REGION Network 10: Stack Door Common Monitoring#7
   RUNG wire#powerrail
      Contact( #TRUE )
      wire#w1
      Contact( "Safety.DataFromSafety".fDoorCoilStatus.anodeWasteDoorUnlock )
      wire#w2
      Coil( "Safetyinterface".StackDoor7.monitoring.DoorOpen )
   END_RUNG
   RUNG wire#w1
      I_Contact( "Safety.DataFromSafety".fDoorCoilStatus.anodeWasteDoorUnlock )
      Contact( "Safety.DataFromSafety".fDoorDrive.fDoor7.ackReq )
      I_Contact( "Global.Data".general.clock.cycle1000Msec )
      I_Contact( "Safety.DataFromSafety".fDoorSwitchStatus.anodeWasteDoorOpen )
   END_RUNG wire#w2
   RUNG wire#w1
      Contact( "Safety.DataFromSafety".fDoorCoilStatus.anodeWasteDoorUnlock )
      Coil( "Safetyinterface".StackDoor7.monitoring.DoorUnLock )
   END_RUNG
   RUNG wire#w1
      I_Contact( "Safety.DataFromSafety".fDoorCoilStatus.anodeWasteDoorUnlock )
      wire#w3
      I_Contact( "Safety.DataFromSafety".fDoorDrive.fDoor7.ackReq )
      wire#w4
      I_Contact( "Safety.DataFromSafety".fDoorSwitchStatus.anodeWasteDoorOpen )
      I_Contact( "Safetyinterface".StackDoor7.monitoring.DoorOpen )
      Coil( "Safetyinterface".StackDoor7.monitoring.DoorClose )
   END_RUNG
   RUNG wire#w3
      Contact( "Safety.DataFromSafety".fDoorDrive.fDoor7.ackReq )
      I_Contact( "Global.Data".general.clock.cycle1000Msec )
   END_RUNG wire#w4
   RUNG wire#w4
      Coil( "Safetyinterface".StackDoor7.monitoring.DoorLock )
   END_RUNG
   // the same network as SCL:
   "Safetyinterface".StackDoor7.monitoring.DoorOpen := #TRUE AND ("Safety.DataFromSafety".fDoorCoilStatus.anodeWasteDoorUnlock OR (NOT "Safety.DataFromSafety".fDoorCoilStatus.anodeWasteDoorUnlock AND "Safety.DataFromSafety".fDoorDrive.fDoor7.ackReq AND NOT "Global.Data".general.clock.cycle1000Msec AND NOT "Safety.DataFromSafety".fDoorSwitchStatus.anodeWasteDoorOpen));
   "Safetyinterface".StackDoor7.monitoring.DoorUnLock := #TRUE AND "Safety.DataFromSafety".fDoorCoilStatus.anodeWasteDoorUnlock;
   #_w1 := #TRUE AND NOT "Safety.DataFromSafety".fDoorCoilStatus.anodeWasteDoorUnlock AND (NOT "Safety.DataFromSafety".fDoorDrive.fDoor7.ackReq OR ("Safety.DataFromSafety".fDoorDrive.fDoor7.ackReq AND NOT "Global.Data".general.clock.cycle1000Msec));
   "Safetyinterface".StackDoor7.monitoring.DoorClose := #_w1 AND NOT "Safety.DataFromSafety".fDoorSwitchStatus.anodeWasteDoorOpen AND NOT "Safetyinterface".StackDoor7.monitoring.DoorOpen;
   "Safetyinterface".StackDoor7.monitoring.DoorLock := #_w1;
END_REGION

REGION Network 11: Stack Door Common Command#8
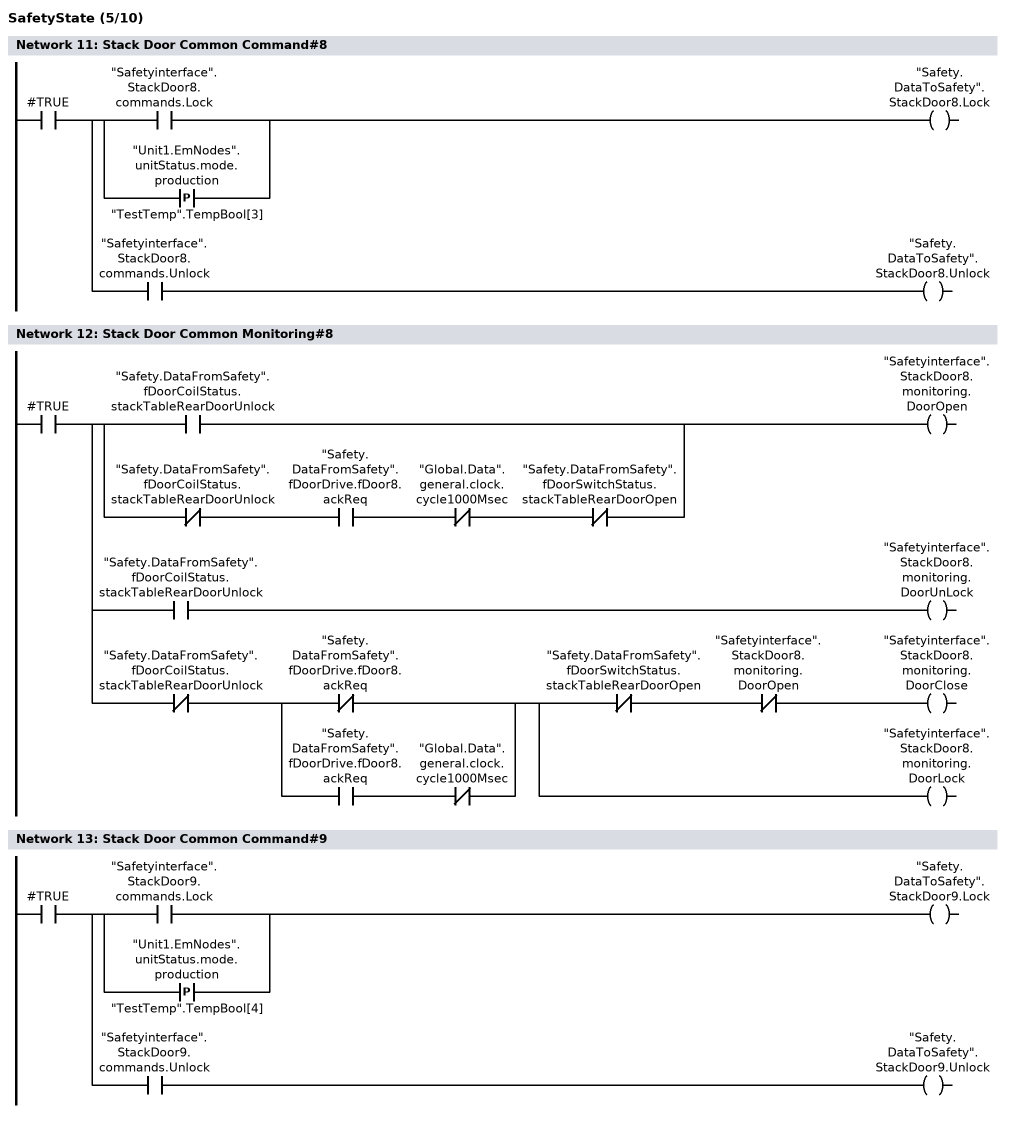
   RUNG wire#powerrail
      Contact( #TRUE )
      wire#w1
      Contact( "Safetyinterface".StackDoor8.commands.Lock )
      wire#w2
      Coil( "Safety.DataToSafety".StackDoor8.Lock )
   END_RUNG
   RUNG wire#w1
      P_Contact(operand := "Unit1.EmNodes".unitStatus.mode.production, bit := "TestTemp".TempBool[3])
   END_RUNG wire#w2
   RUNG wire#w1
      Contact( "Safetyinterface".StackDoor8.commands.Unlock )
      Coil( "Safety.DataToSafety".StackDoor8.Unlock )
   END_RUNG
   // the same network as SCL:
   #_w1 := #TRUE AND "Unit1.EmNodes".unitStatus.mode.production AND NOT "TestTemp".TempBool[3];   // rising edge of "Unit1.EmNodes".unitStatus.mode.production
   "TestTemp".TempBool[3] := "Unit1.EmNodes".unitStatus.mode.production;
   "Safety.DataToSafety".StackDoor8.Lock := (#TRUE AND "Safetyinterface".StackDoor8.commands.Lock) OR #_w1;
   "Safety.DataToSafety".StackDoor8.Unlock := #TRUE AND "Safetyinterface".StackDoor8.commands.Unlock;
END_REGION

REGION Network 12: Stack Door Common Monitoring#8
   RUNG wire#powerrail
      Contact( #TRUE )
      wire#w1
      Contact( "Safety.DataFromSafety".fDoorCoilStatus.stackTableRearDoorUnlock )
      wire#w2
      Coil( "Safetyinterface".StackDoor8.monitoring.DoorOpen )
   END_RUNG
   RUNG wire#w1
      I_Contact( "Safety.DataFromSafety".fDoorCoilStatus.stackTableRearDoorUnlock )
      Contact( "Safety.DataFromSafety".fDoorDrive.fDoor8.ackReq )
      I_Contact( "Global.Data".general.clock.cycle1000Msec )
      I_Contact( "Safety.DataFromSafety".fDoorSwitchStatus.stackTableRearDoorOpen )
   END_RUNG wire#w2
   RUNG wire#w1
      Contact( "Safety.DataFromSafety".fDoorCoilStatus.stackTableRearDoorUnlock )
      Coil( "Safetyinterface".StackDoor8.monitoring.DoorUnLock )
   END_RUNG
   RUNG wire#w1
      I_Contact( "Safety.DataFromSafety".fDoorCoilStatus.stackTableRearDoorUnlock )
      wire#w3
      I_Contact( "Safety.DataFromSafety".fDoorDrive.fDoor8.ackReq )
      wire#w4
      I_Contact( "Safety.DataFromSafety".fDoorSwitchStatus.stackTableRearDoorOpen )
      I_Contact( "Safetyinterface".StackDoor8.monitoring.DoorOpen )
      Coil( "Safetyinterface".StackDoor8.monitoring.DoorClose )
   END_RUNG
   RUNG wire#w3
      Contact( "Safety.DataFromSafety".fDoorDrive.fDoor8.ackReq )
      I_Contact( "Global.Data".general.clock.cycle1000Msec )
   END_RUNG wire#w4
   RUNG wire#w4
      Coil( "Safetyinterface".StackDoor8.monitoring.DoorLock )
   END_RUNG
   // the same network as SCL:
   "Safetyinterface".StackDoor8.monitoring.DoorOpen := #TRUE AND ("Safety.DataFromSafety".fDoorCoilStatus.stackTableRearDoorUnlock OR (NOT "Safety.DataFromSafety".fDoorCoilStatus.stackTableRearDoorUnlock AND "Safety.DataFromSafety".fDoorDrive.fDoor8.ackReq AND NOT "Global.Data".general.clock.cycle1000Msec AND NOT "Safety.DataFromSafety".fDoorSwitchStatus.stackTableRearDoorOpen));
   "Safetyinterface".StackDoor8.monitoring.DoorUnLock := #TRUE AND "Safety.DataFromSafety".fDoorCoilStatus.stackTableRearDoorUnlock;
   #_w1 := #TRUE AND NOT "Safety.DataFromSafety".fDoorCoilStatus.stackTableRearDoorUnlock AND (NOT "Safety.DataFromSafety".fDoorDrive.fDoor8.ackReq OR ("Safety.DataFromSafety".fDoorDrive.fDoor8.ackReq AND NOT "Global.Data".general.clock.cycle1000Msec));
   "Safetyinterface".StackDoor8.monitoring.DoorClose := #_w1 AND NOT "Safety.DataFromSafety".fDoorSwitchStatus.stackTableRearDoorOpen AND NOT "Safetyinterface".StackDoor8.monitoring.DoorOpen;
   "Safetyinterface".StackDoor8.monitoring.DoorLock := #_w1;
END_REGION

REGION Network 13: Stack Door Common Command#9
   RUNG wire#powerrail
      Contact( #TRUE )
      wire#w1
      Contact( "Safetyinterface".StackDoor9.commands.Lock )
      wire#w2
      Coil( "Safety.DataToSafety".StackDoor9.Lock )
   END_RUNG
   RUNG wire#w1
      P_Contact(operand := "Unit1.EmNodes".unitStatus.mode.production, bit := "TestTemp".TempBool[4])
   END_RUNG wire#w2
   RUNG wire#w1
      Contact( "Safetyinterface".StackDoor9.commands.Unlock )
      Coil( "Safety.DataToSafety".StackDoor9.Unlock )
   END_RUNG
   // the same network as SCL:
   #_w1 := #TRUE AND "Unit1.EmNodes".unitStatus.mode.production AND NOT "TestTemp".TempBool[4];   // rising edge of "Unit1.EmNodes".unitStatus.mode.production
   "TestTemp".TempBool[4] := "Unit1.EmNodes".unitStatus.mode.production;
   "Safety.DataToSafety".StackDoor9.Lock := (#TRUE AND "Safetyinterface".StackDoor9.commands.Lock) OR #_w1;
   "Safety.DataToSafety".StackDoor9.Unlock := #TRUE AND "Safetyinterface".StackDoor9.commands.Unlock;
END_REGION

REGION Network 14: Stack Door Common Monitoring#9
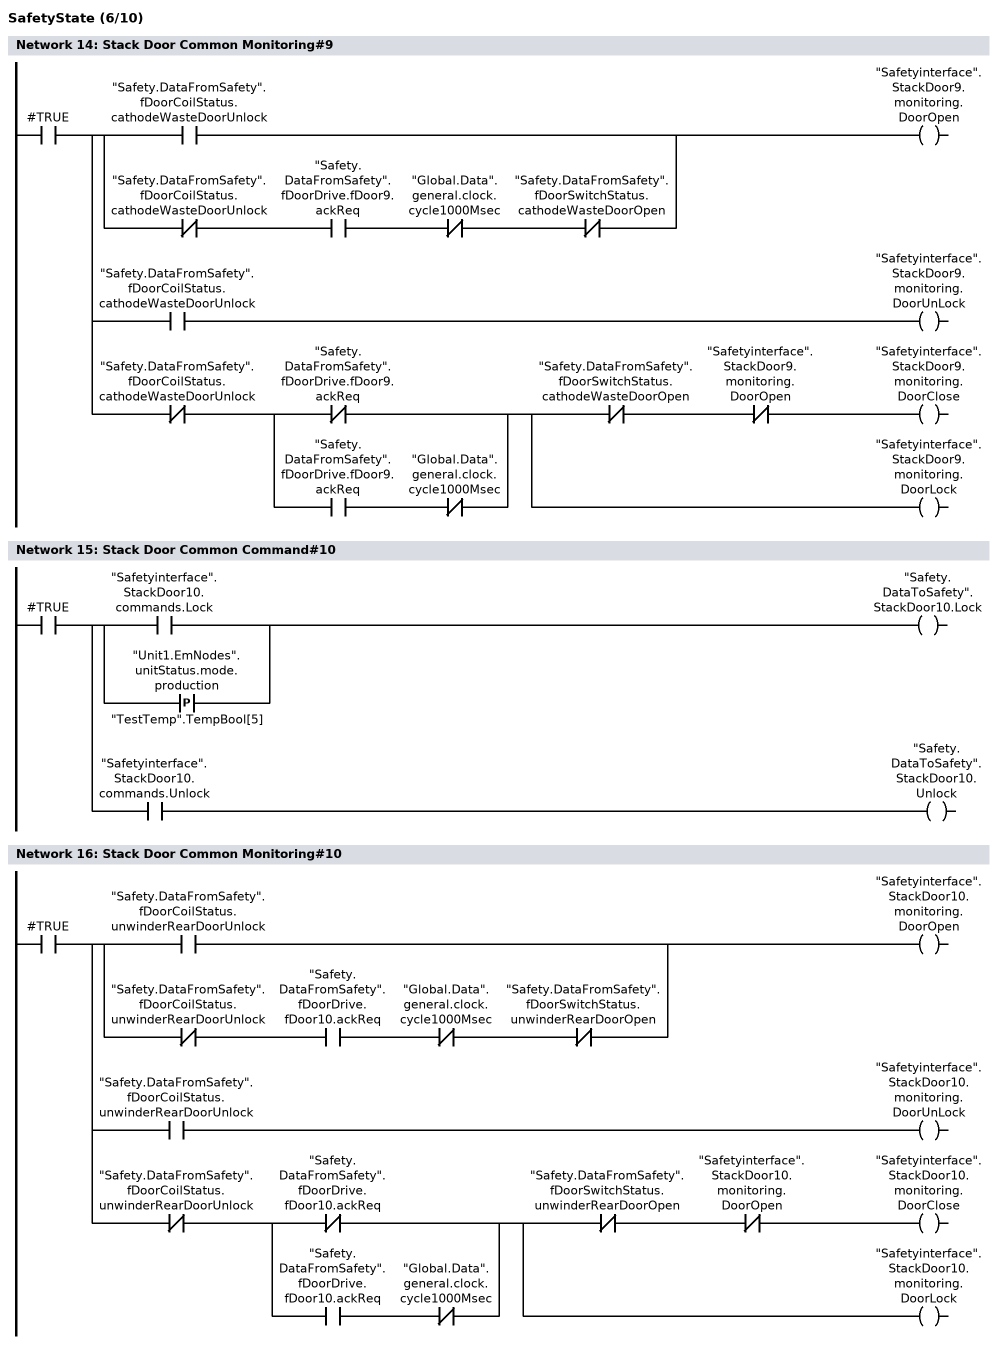
   RUNG wire#powerrail
      Contact( #TRUE )
      wire#w1
      Contact( "Safety.DataFromSafety".fDoorCoilStatus.cathodeWasteDoorUnlock )
      wire#w2
      Coil( "Safetyinterface".StackDoor9.monitoring.DoorOpen )
   END_RUNG
   RUNG wire#w1
      I_Contact( "Safety.DataFromSafety".fDoorCoilStatus.cathodeWasteDoorUnlock )
      Contact( "Safety.DataFromSafety".fDoorDrive.fDoor9.ackReq )
      I_Contact( "Global.Data".general.clock.cycle1000Msec )
      I_Contact( "Safety.DataFromSafety".fDoorSwitchStatus.cathodeWasteDoorOpen )
   END_RUNG wire#w2
   RUNG wire#w1
      Contact( "Safety.DataFromSafety".fDoorCoilStatus.cathodeWasteDoorUnlock )
      Coil( "Safetyinterface".StackDoor9.monitoring.DoorUnLock )
   END_RUNG
   RUNG wire#w1
      I_Contact( "Safety.DataFromSafety".fDoorCoilStatus.cathodeWasteDoorUnlock )
      wire#w3
      I_Contact( "Safety.DataFromSafety".fDoorDrive.fDoor9.ackReq )
      wire#w4
      I_Contact( "Safety.DataFromSafety".fDoorSwitchStatus.cathodeWasteDoorOpen )
      I_Contact( "Safetyinterface".StackDoor9.monitoring.DoorOpen )
      Coil( "Safetyinterface".StackDoor9.monitoring.DoorClose )
   END_RUNG
   RUNG wire#w3
      Contact( "Safety.DataFromSafety".fDoorDrive.fDoor9.ackReq )
      I_Contact( "Global.Data".general.clock.cycle1000Msec )
   END_RUNG wire#w4
   RUNG wire#w4
      Coil( "Safetyinterface".StackDoor9.monitoring.DoorLock )
   END_RUNG
   // the same network as SCL:
   "Safetyinterface".StackDoor9.monitoring.DoorOpen := #TRUE AND ("Safety.DataFromSafety".fDoorCoilStatus.cathodeWasteDoorUnlock OR (NOT "Safety.DataFromSafety".fDoorCoilStatus.cathodeWasteDoorUnlock AND "Safety.DataFromSafety".fDoorDrive.fDoor9.ackReq AND NOT "Global.Data".general.clock.cycle1000Msec AND NOT "Safety.DataFromSafety".fDoorSwitchStatus.cathodeWasteDoorOpen));
   "Safetyinterface".StackDoor9.monitoring.DoorUnLock := #TRUE AND "Safety.DataFromSafety".fDoorCoilStatus.cathodeWasteDoorUnlock;
   #_w1 := #TRUE AND NOT "Safety.DataFromSafety".fDoorCoilStatus.cathodeWasteDoorUnlock AND (NOT "Safety.DataFromSafety".fDoorDrive.fDoor9.ackReq OR ("Safety.DataFromSafety".fDoorDrive.fDoor9.ackReq AND NOT "Global.Data".general.clock.cycle1000Msec));
   "Safetyinterface".StackDoor9.monitoring.DoorClose := #_w1 AND NOT "Safety.DataFromSafety".fDoorSwitchStatus.cathodeWasteDoorOpen AND NOT "Safetyinterface".StackDoor9.monitoring.DoorOpen;
   "Safetyinterface".StackDoor9.monitoring.DoorLock := #_w1;
END_REGION

REGION Network 15: Stack Door Common Command#10
   RUNG wire#powerrail
      Contact( #TRUE )
      wire#w1
      Contact( "Safetyinterface".StackDoor10.commands.Lock )
      wire#w2
      Coil( "Safety.DataToSafety".StackDoor10.Lock )
   END_RUNG
   RUNG wire#w1
      P_Contact(operand := "Unit1.EmNodes".unitStatus.mode.production, bit := "TestTemp".TempBool[5])
   END_RUNG wire#w2
   RUNG wire#w1
      Contact( "Safetyinterface".StackDoor10.commands.Unlock )
      Coil( "Safety.DataToSafety".StackDoor10.Unlock )
   END_RUNG
   // the same network as SCL:
   #_w1 := #TRUE AND "Unit1.EmNodes".unitStatus.mode.production AND NOT "TestTemp".TempBool[5];   // rising edge of "Unit1.EmNodes".unitStatus.mode.production
   "TestTemp".TempBool[5] := "Unit1.EmNodes".unitStatus.mode.production;
   "Safety.DataToSafety".StackDoor10.Lock := (#TRUE AND "Safetyinterface".StackDoor10.commands.Lock) OR #_w1;
   "Safety.DataToSafety".StackDoor10.Unlock := #TRUE AND "Safetyinterface".StackDoor10.commands.Unlock;
END_REGION

REGION Network 16: Stack Door Common Monitoring#10
   RUNG wire#powerrail
      Contact( #TRUE )
      wire#w1
      Contact( "Safety.DataFromSafety".fDoorCoilStatus.unwinderRearDoorUnlock )
      wire#w2
      Coil( "Safetyinterface".StackDoor10.monitoring.DoorOpen )
   END_RUNG
   RUNG wire#w1
      I_Contact( "Safety.DataFromSafety".fDoorCoilStatus.unwinderRearDoorUnlock )
      Contact( "Safety.DataFromSafety".fDoorDrive.fDoor10.ackReq )
      I_Contact( "Global.Data".general.clock.cycle1000Msec )
      I_Contact( "Safety.DataFromSafety".fDoorSwitchStatus.unwinderRearDoorOpen )
   END_RUNG wire#w2
   RUNG wire#w1
      Contact( "Safety.DataFromSafety".fDoorCoilStatus.unwinderRearDoorUnlock )
      Coil( "Safetyinterface".StackDoor10.monitoring.DoorUnLock )
   END_RUNG
   RUNG wire#w1
      I_Contact( "Safety.DataFromSafety".fDoorCoilStatus.unwinderRearDoorUnlock )
      wire#w3
      I_Contact( "Safety.DataFromSafety".fDoorDrive.fDoor10.ackReq )
      wire#w4
      I_Contact( "Safety.DataFromSafety".fDoorSwitchStatus.unwinderRearDoorOpen )
      I_Contact( "Safetyinterface".StackDoor10.monitoring.DoorOpen )
      Coil( "Safetyinterface".StackDoor10.monitoring.DoorClose )
   END_RUNG
   RUNG wire#w3
      Contact( "Safety.DataFromSafety".fDoorDrive.fDoor10.ackReq )
      I_Contact( "Global.Data".general.clock.cycle1000Msec )
   END_RUNG wire#w4
   RUNG wire#w4
      Coil( "Safetyinterface".StackDoor10.monitoring.DoorLock )
   END_RUNG
   // the same network as SCL:
   "Safetyinterface".StackDoor10.monitoring.DoorOpen := #TRUE AND ("Safety.DataFromSafety".fDoorCoilStatus.unwinderRearDoorUnlock OR (NOT "Safety.DataFromSafety".fDoorCoilStatus.unwinderRearDoorUnlock AND "Safety.DataFromSafety".fDoorDrive.fDoor10.ackReq AND NOT "Global.Data".general.clock.cycle1000Msec AND NOT "Safety.DataFromSafety".fDoorSwitchStatus.unwinderRearDoorOpen));
   "Safetyinterface".StackDoor10.monitoring.DoorUnLock := #TRUE AND "Safety.DataFromSafety".fDoorCoilStatus.unwinderRearDoorUnlock;
   #_w1 := #TRUE AND NOT "Safety.DataFromSafety".fDoorCoilStatus.unwinderRearDoorUnlock AND (NOT "Safety.DataFromSafety".fDoorDrive.fDoor10.ackReq OR ("Safety.DataFromSafety".fDoorDrive.fDoor10.ackReq AND NOT "Global.Data".general.clock.cycle1000Msec));
   "Safetyinterface".StackDoor10.monitoring.DoorClose := #_w1 AND NOT "Safety.DataFromSafety".fDoorSwitchStatus.unwinderRearDoorOpen AND NOT "Safetyinterface".StackDoor10.monitoring.DoorOpen;
   "Safetyinterface".StackDoor10.monitoring.DoorLock := #_w1;
END_REGION

REGION Network 17: At Least One Door Unlock Command
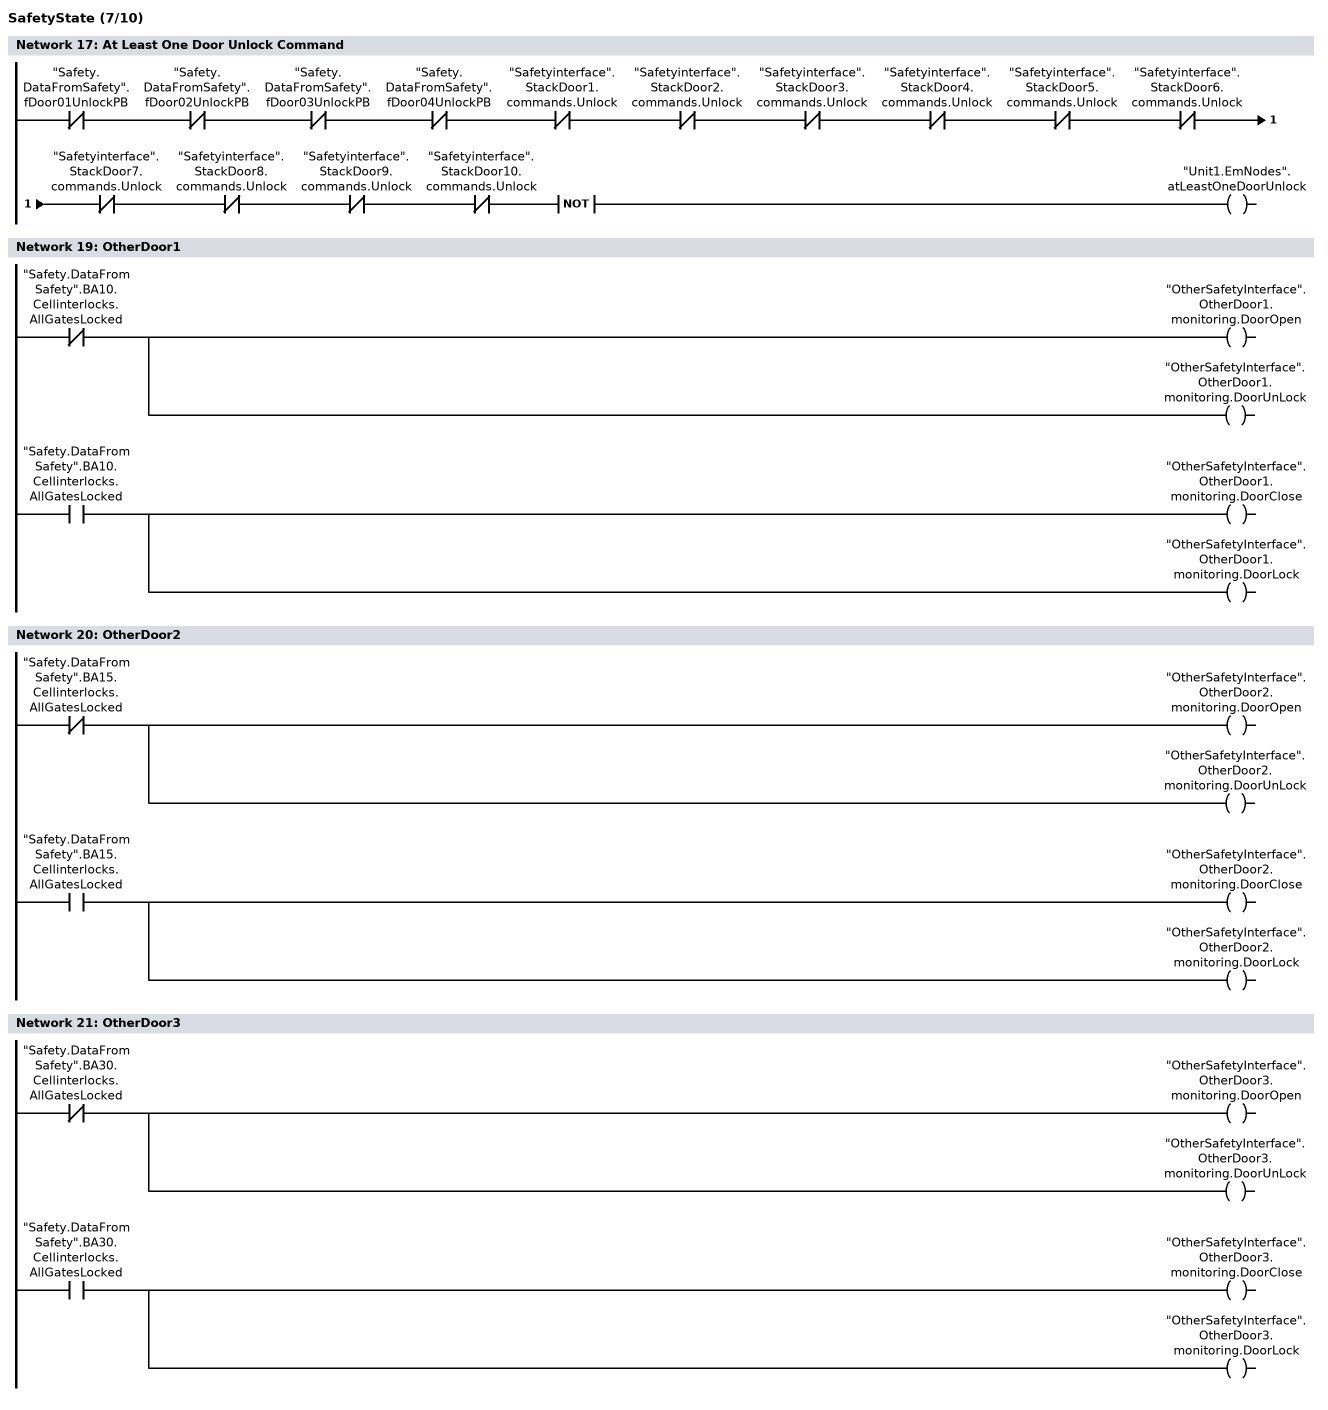
   RUNG wire#powerrail
      I_Contact( "Safety.DataFromSafety".fDoor01UnlockPB )
      I_Contact( "Safety.DataFromSafety".fDoor02UnlockPB )
      I_Contact( "Safety.DataFromSafety".fDoor03UnlockPB )
      I_Contact( "Safety.DataFromSafety".fDoor04UnlockPB )
      I_Contact( "Safetyinterface".StackDoor1.commands.Unlock )
      I_Contact( "Safetyinterface".StackDoor2.commands.Unlock )
      I_Contact( "Safetyinterface".StackDoor3.commands.Unlock )
      I_Contact( "Safetyinterface".StackDoor4.commands.Unlock )
      I_Contact( "Safetyinterface".StackDoor5.commands.Unlock )
      I_Contact( "Safetyinterface".StackDoor6.commands.Unlock )
      I_Contact( "Safetyinterface".StackDoor7.commands.Unlock )
      I_Contact( "Safetyinterface".StackDoor8.commands.Unlock )
      I_Contact( "Safetyinterface".StackDoor9.commands.Unlock )
      I_Contact( "Safetyinterface".StackDoor10.commands.Unlock )
      Not()
      Coil( "Unit1.EmNodes".atLeastOneDoorUnlock )
   END_RUNG
   // the same network as SCL:
   "Unit1.EmNodes".atLeastOneDoorUnlock := NOT (NOT "Safety.DataFromSafety".fDoor01UnlockPB AND NOT "Safety.DataFromSafety".fDoor02UnlockPB AND NOT "Safety.DataFromSafety".fDoor03UnlockPB AND NOT "Safety.DataFromSafety".fDoor04UnlockPB AND NOT "Safetyinterface".StackDoor1.commands.Unlock AND NOT "Safetyinterface".StackDoor2.commands.Unlock AND NOT "Safetyinterface".StackDoor3.commands.Unlock AND NOT "Safetyinterface".StackDoor4.commands.Unlock AND NOT "Safetyinterface".StackDoor5.commands.Unlock AND NOT "Safetyinterface".StackDoor6.commands.Unlock AND NOT "Safetyinterface".StackDoor7.commands.Unlock AND NOT "Safetyinterface".StackDoor8.commands.Unlock AND NOT "Safetyinterface".StackDoor9.commands.Unlock AND NOT "Safetyinterface".StackDoor10.commands.Unlock);
END_REGION

REGION Network 18: ***** Other Safety Interface *****
END_REGION

REGION Network 19: OtherDoor1
   RUNG wire#powerrail
      I_Contact( "Safety.DataFromSafety".BA10.Cellinterlocks.AllGatesLocked )
      wire#w1
      Coil( "OtherSafetyInterface".OtherDoor1.monitoring.DoorOpen )
   END_RUNG
   RUNG wire#w1
      Coil( "OtherSafetyInterface".OtherDoor1.monitoring.DoorUnLock )
   END_RUNG
   RUNG wire#powerrail
      Contact( "Safety.DataFromSafety".BA10.Cellinterlocks.AllGatesLocked )
      wire#w2
      Coil( "OtherSafetyInterface".OtherDoor1.monitoring.DoorClose )
   END_RUNG
   RUNG wire#w2
      Coil( "OtherSafetyInterface".OtherDoor1.monitoring.DoorLock )
   END_RUNG
   // the same network as SCL:
   "OtherSafetyInterface".OtherDoor1.monitoring.DoorOpen := NOT "Safety.DataFromSafety".BA10.Cellinterlocks.AllGatesLocked;
   "OtherSafetyInterface".OtherDoor1.monitoring.DoorUnLock := NOT "Safety.DataFromSafety".BA10.Cellinterlocks.AllGatesLocked;
   "OtherSafetyInterface".OtherDoor1.monitoring.DoorClose := "Safety.DataFromSafety".BA10.Cellinterlocks.AllGatesLocked;
   "OtherSafetyInterface".OtherDoor1.monitoring.DoorLock := "Safety.DataFromSafety".BA10.Cellinterlocks.AllGatesLocked;
END_REGION

REGION Network 20: OtherDoor2
   RUNG wire#powerrail
      I_Contact( "Safety.DataFromSafety".BA15.Cellinterlocks.AllGatesLocked )
      wire#w1
      Coil( "OtherSafetyInterface".OtherDoor2.monitoring.DoorOpen )
   END_RUNG
   RUNG wire#w1
      Coil( "OtherSafetyInterface".OtherDoor2.monitoring.DoorUnLock )
   END_RUNG
   RUNG wire#powerrail
      Contact( "Safety.DataFromSafety".BA15.Cellinterlocks.AllGatesLocked )
      wire#w2
      Coil( "OtherSafetyInterface".OtherDoor2.monitoring.DoorClose )
   END_RUNG
   RUNG wire#w2
      Coil( "OtherSafetyInterface".OtherDoor2.monitoring.DoorLock )
   END_RUNG
   // the same network as SCL:
   "OtherSafetyInterface".OtherDoor2.monitoring.DoorOpen := NOT "Safety.DataFromSafety".BA15.Cellinterlocks.AllGatesLocked;
   "OtherSafetyInterface".OtherDoor2.monitoring.DoorUnLock := NOT "Safety.DataFromSafety".BA15.Cellinterlocks.AllGatesLocked;
   "OtherSafetyInterface".OtherDoor2.monitoring.DoorClose := "Safety.DataFromSafety".BA15.Cellinterlocks.AllGatesLocked;
   "OtherSafetyInterface".OtherDoor2.monitoring.DoorLock := "Safety.DataFromSafety".BA15.Cellinterlocks.AllGatesLocked;
END_REGION

REGION Network 21: OtherDoor3
   RUNG wire#powerrail
      I_Contact( "Safety.DataFromSafety".BA30.Cellinterlocks.AllGatesLocked )
      wire#w1
      Coil( "OtherSafetyInterface".OtherDoor3.monitoring.DoorOpen )
   END_RUNG
   RUNG wire#w1
      Coil( "OtherSafetyInterface".OtherDoor3.monitoring.DoorUnLock )
   END_RUNG
   RUNG wire#powerrail
      Contact( "Safety.DataFromSafety".BA30.Cellinterlocks.AllGatesLocked )
      wire#w2
      Coil( "OtherSafetyInterface".OtherDoor3.monitoring.DoorClose )
   END_RUNG
   RUNG wire#w2
      Coil( "OtherSafetyInterface".OtherDoor3.monitoring.DoorLock )
   END_RUNG
   // the same network as SCL:
   "OtherSafetyInterface".OtherDoor3.monitoring.DoorOpen := NOT "Safety.DataFromSafety".BA30.Cellinterlocks.AllGatesLocked;
   "OtherSafetyInterface".OtherDoor3.monitoring.DoorUnLock := NOT "Safety.DataFromSafety".BA30.Cellinterlocks.AllGatesLocked;
   "OtherSafetyInterface".OtherDoor3.monitoring.DoorClose := "Safety.DataFromSafety".BA30.Cellinterlocks.AllGatesLocked;
   "OtherSafetyInterface".OtherDoor3.monitoring.DoorLock := "Safety.DataFromSafety".BA30.Cellinterlocks.AllGatesLocked;
END_REGION

REGION Network 22: OtherDoor4
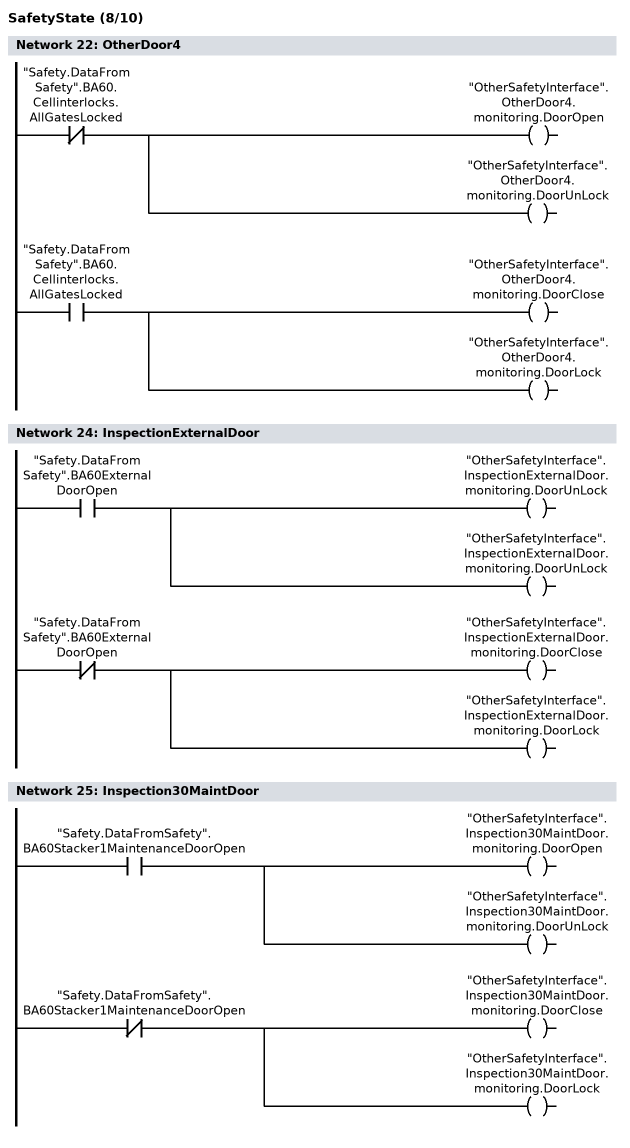
   RUNG wire#powerrail
      I_Contact( "Safety.DataFromSafety".BA60.Cellinterlocks.AllGatesLocked )
      wire#w1
      Coil( "OtherSafetyInterface".OtherDoor4.monitoring.DoorOpen )
   END_RUNG
   RUNG wire#w1
      Coil( "OtherSafetyInterface".OtherDoor4.monitoring.DoorUnLock )
   END_RUNG
   RUNG wire#powerrail
      Contact( "Safety.DataFromSafety".BA60.Cellinterlocks.AllGatesLocked )
      wire#w2
      Coil( "OtherSafetyInterface".OtherDoor4.monitoring.DoorClose )
   END_RUNG
   RUNG wire#w2
      Coil( "OtherSafetyInterface".OtherDoor4.monitoring.DoorLock )
   END_RUNG
   // the same network as SCL:
   "OtherSafetyInterface".OtherDoor4.monitoring.DoorOpen := NOT "Safety.DataFromSafety".BA60.Cellinterlocks.AllGatesLocked;
   "OtherSafetyInterface".OtherDoor4.monitoring.DoorUnLock := NOT "Safety.DataFromSafety".BA60.Cellinterlocks.AllGatesLocked;
   "OtherSafetyInterface".OtherDoor4.monitoring.DoorClose := "Safety.DataFromSafety".BA60.Cellinterlocks.AllGatesLocked;
   "OtherSafetyInterface".OtherDoor4.monitoring.DoorLock := "Safety.DataFromSafety".BA60.Cellinterlocks.AllGatesLocked;
END_REGION

REGION Network 24: InspectionExternalDoor
   RUNG wire#powerrail
      Contact( "Safety.DataFromSafety".BA60ExternalDoorOpen )
      wire#w1
      Coil( "OtherSafetyInterface".InspectionExternalDoor.monitoring.DoorUnLock )
   END_RUNG
   RUNG wire#w1
      Coil( "OtherSafetyInterface".InspectionExternalDoor.monitoring.DoorUnLock )
   END_RUNG
   RUNG wire#powerrail
      I_Contact( "Safety.DataFromSafety".BA60ExternalDoorOpen )
      wire#w2
      Coil( "OtherSafetyInterface".InspectionExternalDoor.monitoring.DoorClose )
   END_RUNG
   RUNG wire#w2
      Coil( "OtherSafetyInterface".InspectionExternalDoor.monitoring.DoorLock )
   END_RUNG
   // the same network as SCL:
   "OtherSafetyInterface".InspectionExternalDoor.monitoring.DoorUnLock := "Safety.DataFromSafety".BA60ExternalDoorOpen;
   "OtherSafetyInterface".InspectionExternalDoor.monitoring.DoorUnLock := "Safety.DataFromSafety".BA60ExternalDoorOpen;
   "OtherSafetyInterface".InspectionExternalDoor.monitoring.DoorClose := NOT "Safety.DataFromSafety".BA60ExternalDoorOpen;
   "OtherSafetyInterface".InspectionExternalDoor.monitoring.DoorLock := NOT "Safety.DataFromSafety".BA60ExternalDoorOpen;
END_REGION

REGION Network 25: Inspection30MaintDoor
   RUNG wire#powerrail
      Contact( "Safety.DataFromSafety".BA60Stacker1MaintenanceDoorOpen )
      wire#w1
      Coil( "OtherSafetyInterface".Inspection30MaintDoor.monitoring.DoorOpen )
   END_RUNG
   RUNG wire#w1
      Coil( "OtherSafetyInterface".Inspection30MaintDoor.monitoring.DoorUnLock )
   END_RUNG
   RUNG wire#powerrail
      I_Contact( "Safety.DataFromSafety".BA60Stacker1MaintenanceDoorOpen )
      wire#w2
      Coil( "OtherSafetyInterface".Inspection30MaintDoor.monitoring.DoorClose )
   END_RUNG
   RUNG wire#w2
      Coil( "OtherSafetyInterface".Inspection30MaintDoor.monitoring.DoorLock )
   END_RUNG
   // the same network as SCL:
   "OtherSafetyInterface".Inspection30MaintDoor.monitoring.DoorOpen := "Safety.DataFromSafety".BA60Stacker1MaintenanceDoorOpen;
   "OtherSafetyInterface".Inspection30MaintDoor.monitoring.DoorUnLock := "Safety.DataFromSafety".BA60Stacker1MaintenanceDoorOpen;
   "OtherSafetyInterface".Inspection30MaintDoor.monitoring.DoorClose := NOT "Safety.DataFromSafety".BA60Stacker1MaintenanceDoorOpen;
   "OtherSafetyInterface".Inspection30MaintDoor.monitoring.DoorLock := NOT "Safety.DataFromSafety".BA60Stacker1MaintenanceDoorOpen;
END_REGION

REGION Network 26: Inspection40MaintDoor
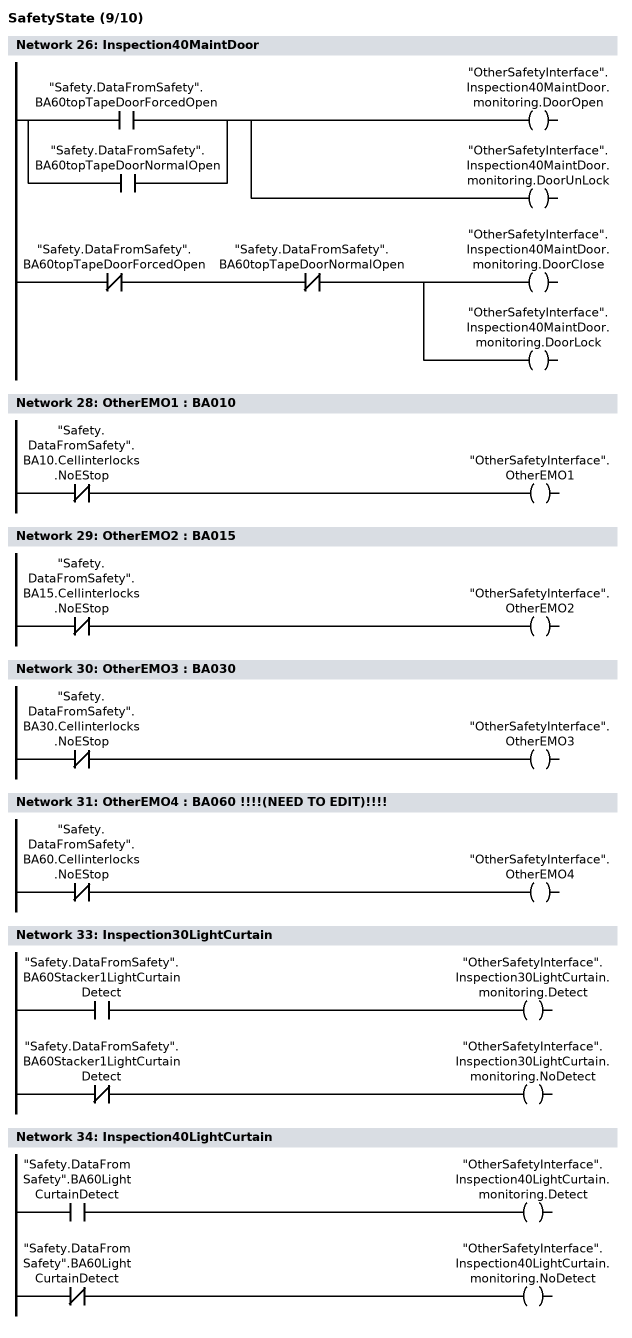
   RUNG wire#powerrail
      Contact( "Safety.DataFromSafety".BA60topTapeDoorForcedOpen )
      wire#w1
      Coil( "OtherSafetyInterface".Inspection40MaintDoor.monitoring.DoorOpen )
   END_RUNG
   RUNG wire#powerrail
      Contact( "Safety.DataFromSafety".BA60topTapeDoorNormalOpen )
   END_RUNG wire#w1
   RUNG wire#w1
      Coil( "OtherSafetyInterface".Inspection40MaintDoor.monitoring.DoorUnLock )
   END_RUNG
   RUNG wire#powerrail
      I_Contact( "Safety.DataFromSafety".BA60topTapeDoorForcedOpen )
      I_Contact( "Safety.DataFromSafety".BA60topTapeDoorNormalOpen )
      wire#w2
      Coil( "OtherSafetyInterface".Inspection40MaintDoor.monitoring.DoorClose )
   END_RUNG
   RUNG wire#w2
      Coil( "OtherSafetyInterface".Inspection40MaintDoor.monitoring.DoorLock )
   END_RUNG
   // the same network as SCL:
   "OtherSafetyInterface".Inspection40MaintDoor.monitoring.DoorOpen := "Safety.DataFromSafety".BA60topTapeDoorForcedOpen OR "Safety.DataFromSafety".BA60topTapeDoorNormalOpen;
   "OtherSafetyInterface".Inspection40MaintDoor.monitoring.DoorUnLock := "OtherSafetyInterface".Inspection40MaintDoor.monitoring.DoorOpen;
   "OtherSafetyInterface".Inspection40MaintDoor.monitoring.DoorClose := NOT "Safety.DataFromSafety".BA60topTapeDoorForcedOpen AND NOT "Safety.DataFromSafety".BA60topTapeDoorNormalOpen;
   "OtherSafetyInterface".Inspection40MaintDoor.monitoring.DoorLock := "OtherSafetyInterface".Inspection40MaintDoor.monitoring.DoorClose;
END_REGION

REGION Network 28: OtherEMO1 : BA010
   RUNG wire#powerrail
      I_Contact( "Safety.DataFromSafety".BA10.Cellinterlocks.NoEStop )
      Coil( "OtherSafetyInterface".OtherEMO1 )
   END_RUNG
   // the same network as SCL:
   "OtherSafetyInterface".OtherEMO1 := NOT "Safety.DataFromSafety".BA10.Cellinterlocks.NoEStop;
END_REGION

REGION Network 29: OtherEMO2 : BA015
   RUNG wire#powerrail
      I_Contact( "Safety.DataFromSafety".BA15.Cellinterlocks.NoEStop )
      Coil( "OtherSafetyInterface".OtherEMO2 )
   END_RUNG
   // the same network as SCL:
   "OtherSafetyInterface".OtherEMO2 := NOT "Safety.DataFromSafety".BA15.Cellinterlocks.NoEStop;
END_REGION

REGION Network 30: OtherEMO3 : BA030
   RUNG wire#powerrail
      I_Contact( "Safety.DataFromSafety".BA30.Cellinterlocks.NoEStop )
      Coil( "OtherSafetyInterface".OtherEMO3 )
   END_RUNG
   // the same network as SCL:
   "OtherSafetyInterface".OtherEMO3 := NOT "Safety.DataFromSafety".BA30.Cellinterlocks.NoEStop;
END_REGION

REGION Network 31: OtherEMO4 : BA060 !!!!(NEED TO EDIT)!!!!
   RUNG wire#powerrail
      I_Contact( "Safety.DataFromSafety".BA60.Cellinterlocks.NoEStop )
      Coil( "OtherSafetyInterface".OtherEMO4 )
   END_RUNG
   // the same network as SCL:
   "OtherSafetyInterface".OtherEMO4 := NOT "Safety.DataFromSafety".BA60.Cellinterlocks.NoEStop;
END_REGION

REGION Network 33: Inspection30LightCurtain
   RUNG wire#powerrail
      Contact( "Safety.DataFromSafety".BA60Stacker1LightCurtainDetect )
      Coil( "OtherSafetyInterface".Inspection30LightCurtain.monitoring.Detect )
   END_RUNG
   RUNG wire#powerrail
      I_Contact( "Safety.DataFromSafety".BA60Stacker1LightCurtainDetect )
      Coil( "OtherSafetyInterface".Inspection30LightCurtain.monitoring.NoDetect )
   END_RUNG
   // the same network as SCL:
   "OtherSafetyInterface".Inspection30LightCurtain.monitoring.Detect := "Safety.DataFromSafety".BA60Stacker1LightCurtainDetect;
   "OtherSafetyInterface".Inspection30LightCurtain.monitoring.NoDetect := NOT "Safety.DataFromSafety".BA60Stacker1LightCurtainDetect;
END_REGION

REGION Network 34: Inspection40LightCurtain
   RUNG wire#powerrail
      Contact( "Safety.DataFromSafety".BA60LightCurtainDetect )
      Coil( "OtherSafetyInterface".Inspection40LightCurtain.monitoring.Detect )
   END_RUNG
   RUNG wire#powerrail
      I_Contact( "Safety.DataFromSafety".BA60LightCurtainDetect )
      Coil( "OtherSafetyInterface".Inspection40LightCurtain.monitoring.NoDetect )
   END_RUNG
   // the same network as SCL:
   "OtherSafetyInterface".Inspection40LightCurtain.monitoring.Detect := "Safety.DataFromSafety".BA60LightCurtainDetect;
   "OtherSafetyInterface".Inspection40LightCurtain.monitoring.NoDetect := NOT "Safety.DataFromSafety".BA60LightCurtainDetect;
END_REGION

REGION Network 36: 30CathodeConveyorCover
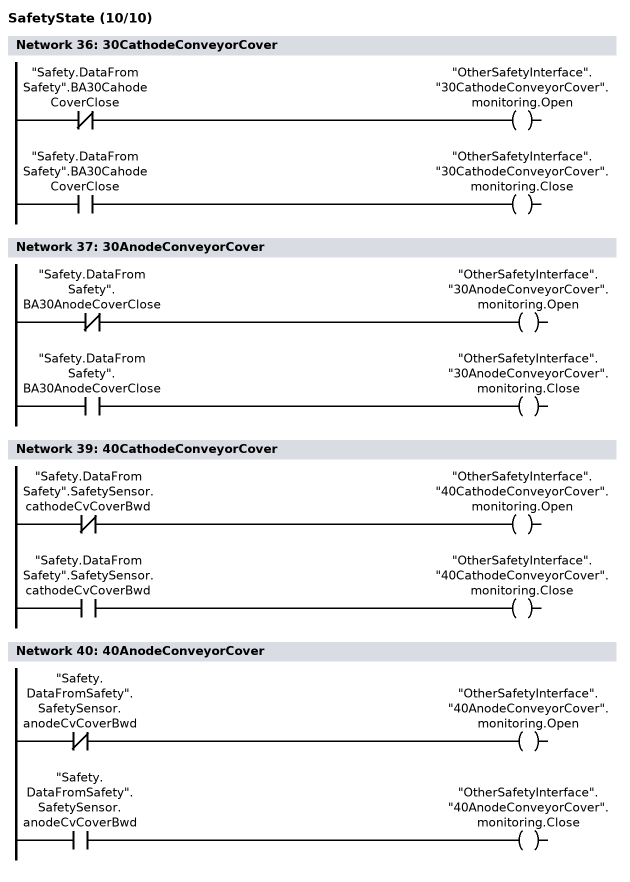
   RUNG wire#powerrail
      I_Contact( "Safety.DataFromSafety".BA30CahodeCoverClose )
      Coil( "OtherSafetyInterface"."30CathodeConveyorCover".monitoring.Open )
   END_RUNG
   RUNG wire#powerrail
      Contact( "Safety.DataFromSafety".BA30CahodeCoverClose )
      Coil( "OtherSafetyInterface"."30CathodeConveyorCover".monitoring.Close )
   END_RUNG
   // the same network as SCL:
   "OtherSafetyInterface"."30CathodeConveyorCover".monitoring.Open := NOT "Safety.DataFromSafety".BA30CahodeCoverClose;
   "OtherSafetyInterface"."30CathodeConveyorCover".monitoring.Close := "Safety.DataFromSafety".BA30CahodeCoverClose;
END_REGION

REGION Network 37: 30AnodeConveyorCover
   RUNG wire#powerrail
      I_Contact( "Safety.DataFromSafety".BA30AnodeCoverClose )
      Coil( "OtherSafetyInterface"."30AnodeConveyorCover".monitoring.Open )
   END_RUNG
   RUNG wire#powerrail
      Contact( "Safety.DataFromSafety".BA30AnodeCoverClose )
      Coil( "OtherSafetyInterface"."30AnodeConveyorCover".monitoring.Close )
   END_RUNG
   // the same network as SCL:
   "OtherSafetyInterface"."30AnodeConveyorCover".monitoring.Open := NOT "Safety.DataFromSafety".BA30AnodeCoverClose;
   "OtherSafetyInterface"."30AnodeConveyorCover".monitoring.Close := "Safety.DataFromSafety".BA30AnodeCoverClose;
END_REGION

REGION Network 39: 40CathodeConveyorCover
   RUNG wire#powerrail
      I_Contact( "Safety.DataFromSafety".SafetySensor.cathodeCvCoverBwd )
      Coil( "OtherSafetyInterface"."40CathodeConveyorCover".monitoring.Open )
   END_RUNG
   RUNG wire#powerrail
      Contact( "Safety.DataFromSafety".SafetySensor.cathodeCvCoverBwd )
      Coil( "OtherSafetyInterface"."40CathodeConveyorCover".monitoring.Close )
   END_RUNG
   // the same network as SCL:
   "OtherSafetyInterface"."40CathodeConveyorCover".monitoring.Open := NOT "Safety.DataFromSafety".SafetySensor.cathodeCvCoverBwd;
   "OtherSafetyInterface"."40CathodeConveyorCover".monitoring.Close := "Safety.DataFromSafety".SafetySensor.cathodeCvCoverBwd;
END_REGION

REGION Network 40: 40AnodeConveyorCover
   RUNG wire#powerrail
      I_Contact( "Safety.DataFromSafety".SafetySensor.anodeCvCoverBwd )
      Coil( "OtherSafetyInterface"."40AnodeConveyorCover".monitoring.Open )
   END_RUNG
   RUNG wire#powerrail
      Contact( "Safety.DataFromSafety".SafetySensor.anodeCvCoverBwd )
      Coil( "OtherSafetyInterface"."40AnodeConveyorCover".monitoring.Close )
   END_RUNG
   // the same network as SCL:
   "OtherSafetyInterface"."40AnodeConveyorCover".monitoring.Open := NOT "Safety.DataFromSafety".SafetySensor.anodeCvCoverBwd;
   "OtherSafetyInterface"."40AnodeConveyorCover".monitoring.Close := "Safety.DataFromSafety".SafetySensor.anodeCvCoverBwd;
END_REGION
END_FUNCTION

FUNCTION "CallProductionData" : Void   // FC151, LAD
TITLE = Produktions Daten / Production data
AUTHOR : SICAR
FAMILY : ProdData
VERSION : 1.0
// Dieser Baustein dient als Aufrufschnittstelle für die Funktionsbausteine  
// * _Shiftmodel  
// * _ProdDataCycleTimer  
// * _ProdDataCounter  
// * _ProdDataLimitValues  
// * _ProdDataShiftCounter  
// oder  
// * _ProdDataShiftCounterOee, ShiftProductionTimes
// Call of  FC ProductDataSimulation and LSicar Production Blocks
// stored: IsIECCheckEnabled true, SetENOAutomatically true
   // Ret_Val : Ret_Val
   VAR_TEMP   // added for the SCL form of the ladder/FBD networks
      _w1 : Bool;
      _w2 : Bool;
      _w3 : Bool;
      _w4 : Bool;
      _w5 : Bool;
      _w6 : Bool;
   END_VAR
BEGIN

REGION Network 1: BLOCK INFO HEADER
   // SIEMENS AG / (c)Copyright 2023
   // ------------------------------------------------------------------------------
   // Title:            CallProductionData(FC151)
   // Comment/Function: Call of  FC ProductDataSimulation and LSicar Production Blocks
   // Library/Family:   Automation Framework
   // Author:           Siemens Digital Industry
   // Tested with:      ---
   // Engineering:      TIA Portal V19
   // Restrictions:     -
   // Requirements:     ---
   // ------------------------------------------------------------------------------
   // Change log table:
   // Version  | Date       | Expert in charge       | Changes applied
   // ---------|------------|------------------------|------------------------------
   // 01.00.00 | 11.12.2023 | Siemens Industry Online Support
   //                         First released version
END_REGION

REGION Network 2: Beschreibung / DESCRIPTION
   // **Aufrufschnittstelle**  
   // Der Baustein wird einmalig im zyklischen Programm aufgerufen.  
   // 
   // 
   // #### Weitere Hinweise
   // 
   // #### Updateinfo
   // 
   // #### Weitere Dokumente
   // 
   // ![Icon](_Icon/reference.PNG)
   // 
   // Siehe:  
   // ..\Library Types\LSicar_Shiftmodel.pdf  
   // ..\Library Types\LSicar_ProdDataCycleTimer.pdf  
   // ..\Library Types\LSicar_ProdDataCounter.pdf  
   // ..\Library Types\LSicar_ProdDataLimitValues.pdf  
   // ..\Library Types\LSicar_ProdDataShiftCounter.pdf  
   // ..\Library Types\LSicar_ProdDataShiftCounterOee.pdf  
   // ..\Library Types\LSicar_ShiftProductionTimes.pdf
   // The block is used as a calling interface for the function blocks  
   // *   _Shiftmodel
   // *   _ProdDataCycleTimer
   // *   _ProdDataCounter
   // *   _ProdDataLimitValues
   // *   _ProdDataShiftCounter
   // or
   // *   _ProdDataShiftCounterOee, ShiftProductionTimes
   // 
   // **Calling interface**  
   // The block must be called once only in the cyclic program.  
   // 
   // The block is used as a calling interface for the function blocks  
   // *   _Shiftmodel
   // *   _ProdDataCycleTimer
   // *   _ProdDataCounter
   // *   _ProdDataLimitValues
   // *   _ProdDataShiftCounter
   // or
   // *   _ProdDataShiftCounterOee, ShiftProductionTimes
   // 
   // #### Additional information
   // 
   // #### Update info
   // 
   // #### Further documentations
   // 
   // ![Icon](_Icon/reference.PNG) 
   // 
   // See:  
   // ..\Library Types\LSicar_Shiftmodel.pdf  
   // ..\Library Types\LSicar_ProdDataCycleTimer.pdf  
   // ..\Library Types\LSicar_ProdDataCounter.pdf  
   // ..\Library Types\LSicar_ProdDataLimitValues.pdf  
   // ..\Library Types\LSicar_ProdDataShiftCounter.pdf  
   // ..\Library Types\LSicar_ProdDataShiftCounterOee.pdf  
   // ..\Library Types\LSicar_ShiftProductionTimes.pdf
END_REGION

REGION Network 3: Call Production Simulation
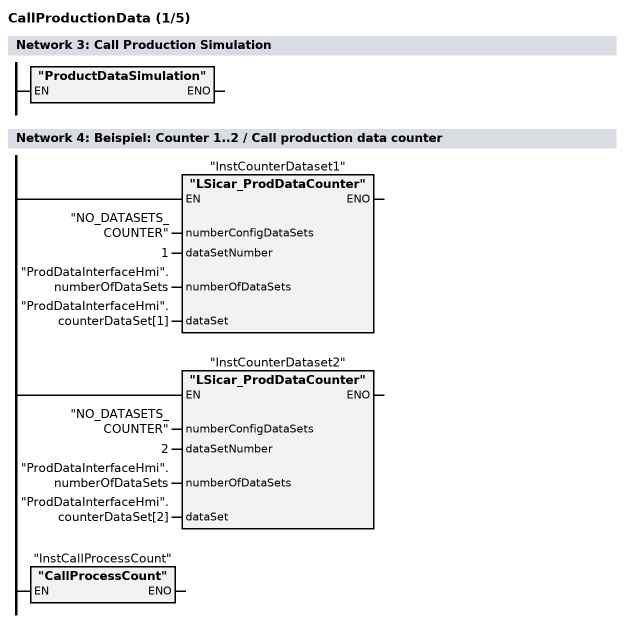
   RUNG wire#powerrail
      "ProductDataSimulation"()
   END_RUNG
   // the same network as SCL:
   "ProductDataSimulation"();
END_REGION

REGION Network 4: Beispiel: Counter 1..2 / Call production data counter
   RUNG wire#powerrail
      "InstCounterDataset1"(numberConfigDataSets := "NO_DATASETS_COUNTER", dataSetNumber := 1, numberOfDataSets := "ProdDataInterfaceHmi".numberOfDataSets, dataSet := "ProdDataInterfaceHmi".counterDataSet[1])
   END_RUNG
   RUNG wire#powerrail
      "InstCounterDataset2"(numberConfigDataSets := "NO_DATASETS_COUNTER", dataSetNumber := 2, numberOfDataSets := "ProdDataInterfaceHmi".numberOfDataSets, dataSet := "ProdDataInterfaceHmi".counterDataSet[2])
   END_RUNG
   RUNG wire#powerrail
      "InstCallProcessCount"()
   END_RUNG
   // the same network as SCL:
   "InstCounterDataset1"(numberConfigDataSets := "NO_DATASETS_COUNTER",   // "LSicar_ProdDataCounter"
                         dataSetNumber := 1,
                         numberOfDataSets := "ProdDataInterfaceHmi".numberOfDataSets,
                         dataSet := "ProdDataInterfaceHmi".counterDataSet[1]);
   "InstCounterDataset2"(numberConfigDataSets := "NO_DATASETS_COUNTER",   // "LSicar_ProdDataCounter"
                         dataSetNumber := 2,
                         numberOfDataSets := "ProdDataInterfaceHmi".numberOfDataSets,
                         dataSet := "ProdDataInterfaceHmi".counterDataSet[2]);
   "InstCallProcessCount"();   // "CallProcessCount"
END_REGION

REGION Network 5: Call production data cycle timer
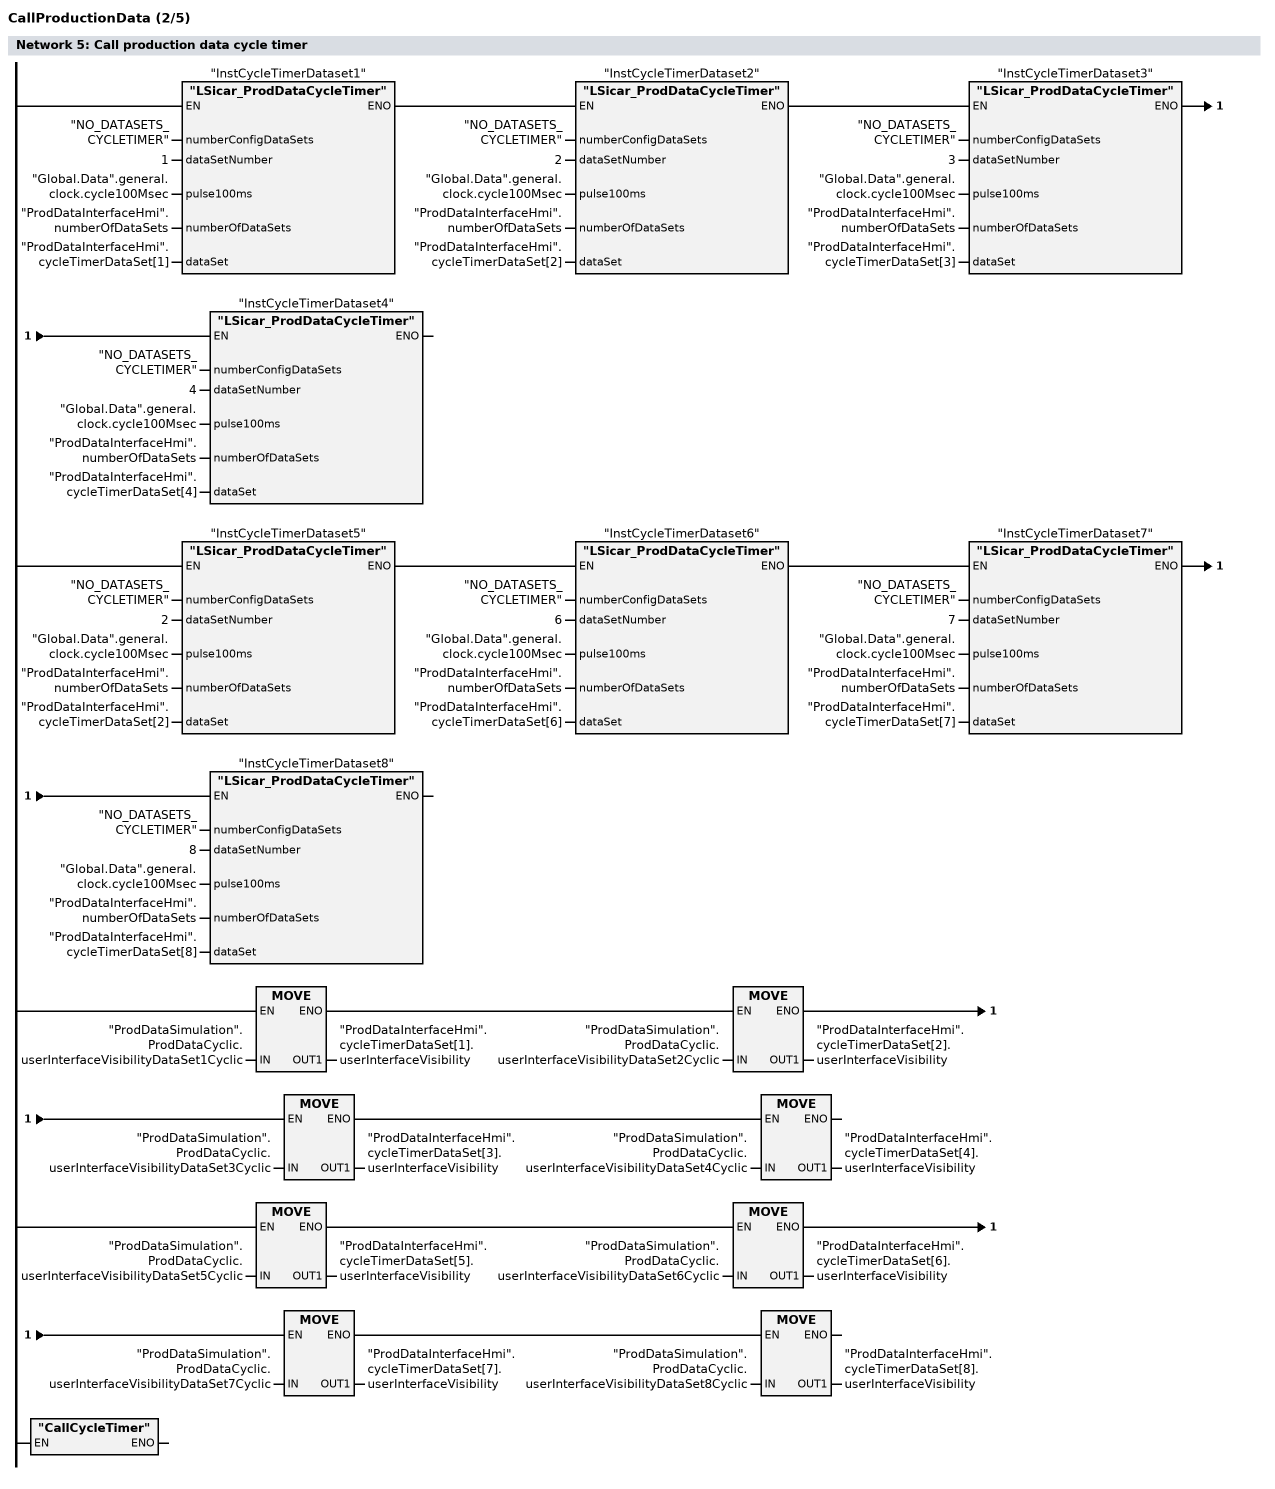
   RUNG wire#powerrail
      "InstCycleTimerDataset1"(numberConfigDataSets := "NO_DATASETS_CYCLETIMER", dataSetNumber := 1, pulse100ms := "Global.Data".general.clock.cycle100Msec, numberOfDataSets := "ProdDataInterfaceHmi".numberOfDataSets, dataSet := "ProdDataInterfaceHmi".cycleTimerDataSet[1])
      "InstCycleTimerDataset2"(numberConfigDataSets := "NO_DATASETS_CYCLETIMER", dataSetNumber := 2, pulse100ms := "Global.Data".general.clock.cycle100Msec, numberOfDataSets := "ProdDataInterfaceHmi".numberOfDataSets, dataSet := "ProdDataInterfaceHmi".cycleTimerDataSet[2])
      "InstCycleTimerDataset3"(numberConfigDataSets := "NO_DATASETS_CYCLETIMER", dataSetNumber := 3, pulse100ms := "Global.Data".general.clock.cycle100Msec, numberOfDataSets := "ProdDataInterfaceHmi".numberOfDataSets, dataSet := "ProdDataInterfaceHmi".cycleTimerDataSet[3])
      "InstCycleTimerDataset4"(numberConfigDataSets := "NO_DATASETS_CYCLETIMER", dataSetNumber := 4, pulse100ms := "Global.Data".general.clock.cycle100Msec, numberOfDataSets := "ProdDataInterfaceHmi".numberOfDataSets, dataSet := "ProdDataInterfaceHmi".cycleTimerDataSet[4])
   END_RUNG
   RUNG wire#powerrail
      "InstCycleTimerDataset5"(numberConfigDataSets := "NO_DATASETS_CYCLETIMER", dataSetNumber := 2, pulse100ms := "Global.Data".general.clock.cycle100Msec, numberOfDataSets := "ProdDataInterfaceHmi".numberOfDataSets, dataSet := "ProdDataInterfaceHmi".cycleTimerDataSet[2])
      "InstCycleTimerDataset6"(numberConfigDataSets := "NO_DATASETS_CYCLETIMER", dataSetNumber := 6, pulse100ms := "Global.Data".general.clock.cycle100Msec, numberOfDataSets := "ProdDataInterfaceHmi".numberOfDataSets, dataSet := "ProdDataInterfaceHmi".cycleTimerDataSet[6])
      "InstCycleTimerDataset7"(numberConfigDataSets := "NO_DATASETS_CYCLETIMER", dataSetNumber := 7, pulse100ms := "Global.Data".general.clock.cycle100Msec, numberOfDataSets := "ProdDataInterfaceHmi".numberOfDataSets, dataSet := "ProdDataInterfaceHmi".cycleTimerDataSet[7])
      "InstCycleTimerDataset8"(numberConfigDataSets := "NO_DATASETS_CYCLETIMER", dataSetNumber := 8, pulse100ms := "Global.Data".general.clock.cycle100Msec, numberOfDataSets := "ProdDataInterfaceHmi".numberOfDataSets, dataSet := "ProdDataInterfaceHmi".cycleTimerDataSet[8])
   END_RUNG
   RUNG wire#powerrail
      Move(in := "ProdDataSimulation".ProdDataCyclic.userInterfaceVisibilityDataSet1Cyclic, out1 => "ProdDataInterfaceHmi".cycleTimerDataSet[1].userInterfaceVisibility)
      Move(in := "ProdDataSimulation".ProdDataCyclic.userInterfaceVisibilityDataSet2Cyclic, out1 => "ProdDataInterfaceHmi".cycleTimerDataSet[2].userInterfaceVisibility)
      Move(in := "ProdDataSimulation".ProdDataCyclic.userInterfaceVisibilityDataSet3Cyclic, out1 => "ProdDataInterfaceHmi".cycleTimerDataSet[3].userInterfaceVisibility)
      Move(in := "ProdDataSimulation".ProdDataCyclic.userInterfaceVisibilityDataSet4Cyclic, out1 => "ProdDataInterfaceHmi".cycleTimerDataSet[4].userInterfaceVisibility)
   END_RUNG
   RUNG wire#powerrail
      Move(in := "ProdDataSimulation".ProdDataCyclic.userInterfaceVisibilityDataSet5Cyclic, out1 => "ProdDataInterfaceHmi".cycleTimerDataSet[5].userInterfaceVisibility)
      Move(in := "ProdDataSimulation".ProdDataCyclic.userInterfaceVisibilityDataSet6Cyclic, out1 => "ProdDataInterfaceHmi".cycleTimerDataSet[6].userInterfaceVisibility)
      Move(in := "ProdDataSimulation".ProdDataCyclic.userInterfaceVisibilityDataSet7Cyclic, out1 => "ProdDataInterfaceHmi".cycleTimerDataSet[7].userInterfaceVisibility)
      Move(in := "ProdDataSimulation".ProdDataCyclic.userInterfaceVisibilityDataSet8Cyclic, out1 => "ProdDataInterfaceHmi".cycleTimerDataSet[8].userInterfaceVisibility)
   END_RUNG
   RUNG wire#powerrail
      "CallCycleTimer"()
   END_RUNG
   // the same network as SCL:
   "InstCycleTimerDataset1"(numberConfigDataSets := "NO_DATASETS_CYCLETIMER",   // "LSicar_ProdDataCycleTimer"
                           dataSetNumber := 1,
                           pulse100ms := "Global.Data".general.clock.cycle100Msec,
                           numberOfDataSets := "ProdDataInterfaceHmi".numberOfDataSets,
                           dataSet := "ProdDataInterfaceHmi".cycleTimerDataSet[1],
                           ENO => #_w1);
   "InstCycleTimerDataset2"(EN := #_w1,   // "LSicar_ProdDataCycleTimer"
                           numberConfigDataSets := "NO_DATASETS_CYCLETIMER",
                           dataSetNumber := 2,
                           pulse100ms := "Global.Data".general.clock.cycle100Msec,
                           numberOfDataSets := "ProdDataInterfaceHmi".numberOfDataSets,
                           dataSet := "ProdDataInterfaceHmi".cycleTimerDataSet[2],
                           ENO => #_w2);
   "InstCycleTimerDataset3"(EN := #_w2,   // "LSicar_ProdDataCycleTimer"
                           numberConfigDataSets := "NO_DATASETS_CYCLETIMER",
                           dataSetNumber := 3,
                           pulse100ms := "Global.Data".general.clock.cycle100Msec,
                           numberOfDataSets := "ProdDataInterfaceHmi".numberOfDataSets,
                           dataSet := "ProdDataInterfaceHmi".cycleTimerDataSet[3],
                           ENO => #_w3);
   IF #_w3 THEN
       "InstCycleTimerDataset4"(numberConfigDataSets := "NO_DATASETS_CYCLETIMER",   // "LSicar_ProdDataCycleTimer"
                               dataSetNumber := 4,
                               pulse100ms := "Global.Data".general.clock.cycle100Msec,
                               numberOfDataSets := "ProdDataInterfaceHmi".numberOfDataSets,
                               dataSet := "ProdDataInterfaceHmi".cycleTimerDataSet[4]);
   END_IF;
   "InstCycleTimerDataset5"(numberConfigDataSets := "NO_DATASETS_CYCLETIMER",   // "LSicar_ProdDataCycleTimer"
                           dataSetNumber := 2,
                           pulse100ms := "Global.Data".general.clock.cycle100Msec,
                           numberOfDataSets := "ProdDataInterfaceHmi".numberOfDataSets,
                           dataSet := "ProdDataInterfaceHmi".cycleTimerDataSet[2],
                           ENO => #_w4);
   "InstCycleTimerDataset6"(EN := #_w4,   // "LSicar_ProdDataCycleTimer"
                           numberConfigDataSets := "NO_DATASETS_CYCLETIMER",
                           dataSetNumber := 6,
                           pulse100ms := "Global.Data".general.clock.cycle100Msec,
                           numberOfDataSets := "ProdDataInterfaceHmi".numberOfDataSets,
                           dataSet := "ProdDataInterfaceHmi".cycleTimerDataSet[6],
                           ENO => #_w5);
   "InstCycleTimerDataset7"(EN := #_w5,   // "LSicar_ProdDataCycleTimer"
                           numberConfigDataSets := "NO_DATASETS_CYCLETIMER",
                           dataSetNumber := 7,
                           pulse100ms := "Global.Data".general.clock.cycle100Msec,
                           numberOfDataSets := "ProdDataInterfaceHmi".numberOfDataSets,
                           dataSet := "ProdDataInterfaceHmi".cycleTimerDataSet[7],
                           ENO => #_w6);
   IF #_w6 THEN
       "InstCycleTimerDataset8"(numberConfigDataSets := "NO_DATASETS_CYCLETIMER",   // "LSicar_ProdDataCycleTimer"
                               dataSetNumber := 8,
                               pulse100ms := "Global.Data".general.clock.cycle100Msec,
                               numberOfDataSets := "ProdDataInterfaceHmi".numberOfDataSets,
                               dataSet := "ProdDataInterfaceHmi".cycleTimerDataSet[8]);
   END_IF;
   "ProdDataInterfaceHmi".cycleTimerDataSet[1].userInterfaceVisibility := "ProdDataSimulation".ProdDataCyclic.userInterfaceVisibilityDataSet1Cyclic;
   "ProdDataInterfaceHmi".cycleTimerDataSet[2].userInterfaceVisibility := "ProdDataSimulation".ProdDataCyclic.userInterfaceVisibilityDataSet2Cyclic;
   "ProdDataInterfaceHmi".cycleTimerDataSet[3].userInterfaceVisibility := "ProdDataSimulation".ProdDataCyclic.userInterfaceVisibilityDataSet3Cyclic;
   "ProdDataInterfaceHmi".cycleTimerDataSet[4].userInterfaceVisibility := "ProdDataSimulation".ProdDataCyclic.userInterfaceVisibilityDataSet4Cyclic;
   "ProdDataInterfaceHmi".cycleTimerDataSet[5].userInterfaceVisibility := "ProdDataSimulation".ProdDataCyclic.userInterfaceVisibilityDataSet5Cyclic;
   "ProdDataInterfaceHmi".cycleTimerDataSet[6].userInterfaceVisibility := "ProdDataSimulation".ProdDataCyclic.userInterfaceVisibilityDataSet6Cyclic;
   "ProdDataInterfaceHmi".cycleTimerDataSet[7].userInterfaceVisibility := "ProdDataSimulation".ProdDataCyclic.userInterfaceVisibilityDataSet7Cyclic;
   "ProdDataInterfaceHmi".cycleTimerDataSet[8].userInterfaceVisibility := "ProdDataSimulation".ProdDataCyclic.userInterfaceVisibilityDataSet8Cyclic;
   "CallCycleTimer"();
END_REGION

REGION Network 6: Beispiel: Limit Value 1..2 / Call production data limit values
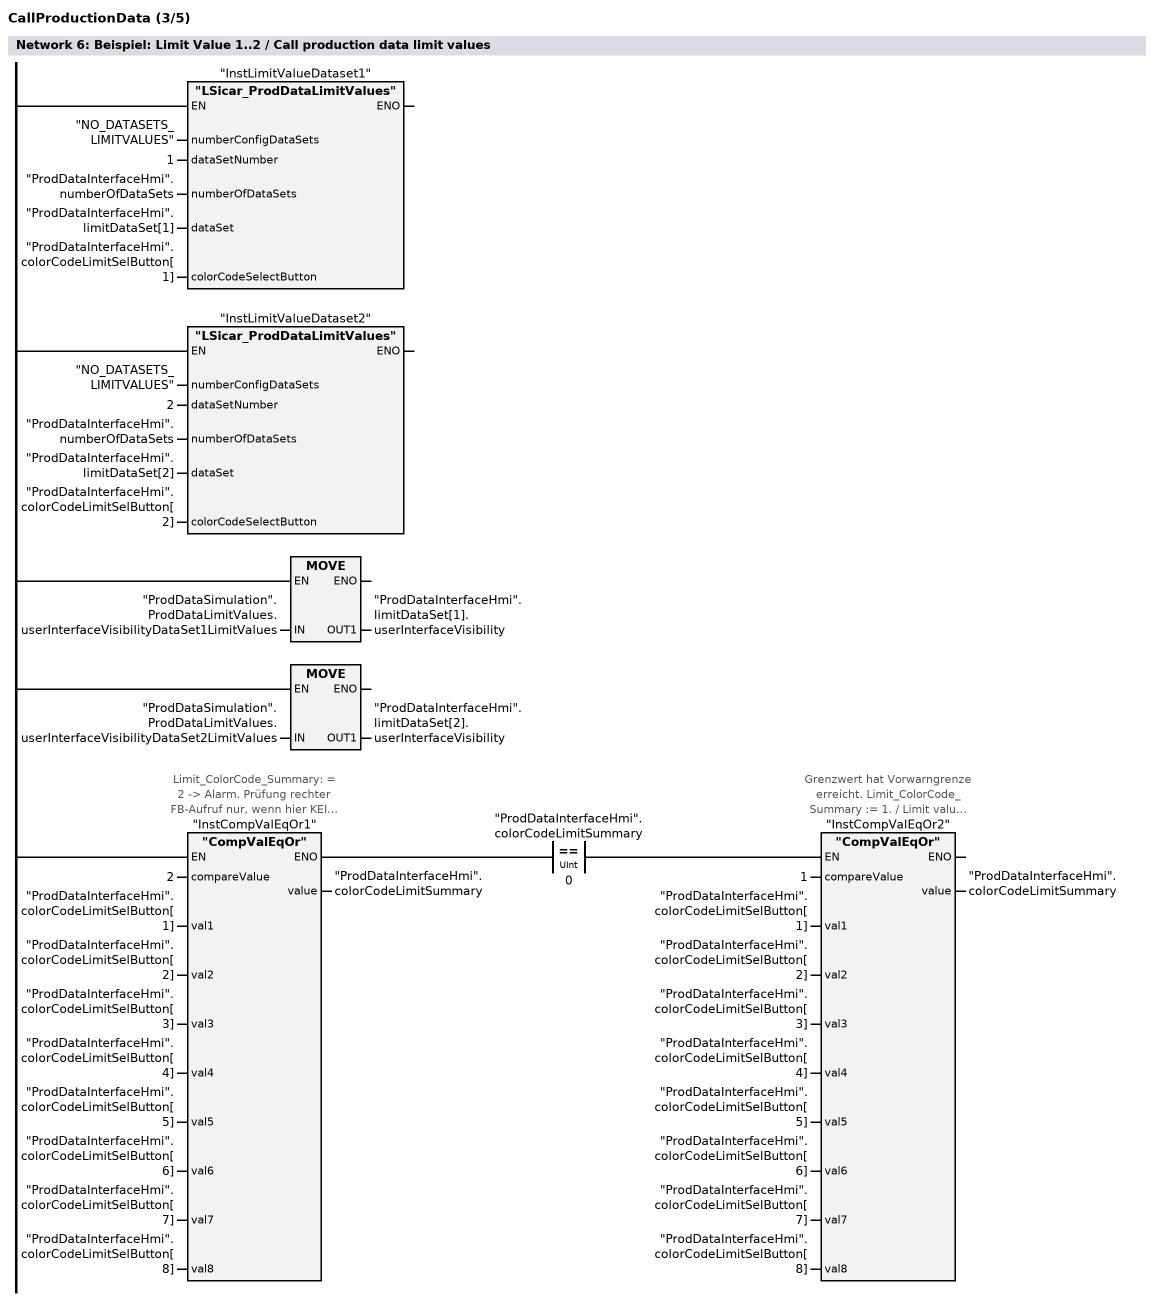
   RUNG wire#powerrail
      "InstLimitValueDataset1"(numberConfigDataSets := "NO_DATASETS_LIMITVALUES", dataSetNumber := 1, numberOfDataSets := "ProdDataInterfaceHmi".numberOfDataSets, dataSet := "ProdDataInterfaceHmi".limitDataSet[1], colorCodeSelectButton := "ProdDataInterfaceHmi".colorCodeLimitSelButton[1])
   END_RUNG
   RUNG wire#powerrail
      "InstLimitValueDataset2"(numberConfigDataSets := "NO_DATASETS_LIMITVALUES", dataSetNumber := 2, numberOfDataSets := "ProdDataInterfaceHmi".numberOfDataSets, dataSet := "ProdDataInterfaceHmi".limitDataSet[2], colorCodeSelectButton := "ProdDataInterfaceHmi".colorCodeLimitSelButton[2])
   END_RUNG
   RUNG wire#powerrail
      Move(in := "ProdDataSimulation".ProdDataLimitValues.userInterfaceVisibilityDataSet1LimitValues, out1 => "ProdDataInterfaceHmi".limitDataSet[1].userInterfaceVisibility)
   END_RUNG
   RUNG wire#powerrail
      Move(in := "ProdDataSimulation".ProdDataLimitValues.userInterfaceVisibilityDataSet2LimitValues, out1 => "ProdDataInterfaceHmi".limitDataSet[2].userInterfaceVisibility)
   END_RUNG
   RUNG wire#powerrail
      "InstCompValEqOr1"(compareValue := 2, val1 := "ProdDataInterfaceHmi".colorCodeLimitSelButton[1], val2 := "ProdDataInterfaceHmi".colorCodeLimitSelButton[2], val3 := "ProdDataInterfaceHmi".colorCodeLimitSelButton[3], val4 := "ProdDataInterfaceHmi".colorCodeLimitSelButton[4], val5 := "ProdDataInterfaceHmi".colorCodeLimitSelButton[5], val6 := "ProdDataInterfaceHmi".colorCodeLimitSelButton[6], val7 := "ProdDataInterfaceHmi".colorCodeLimitSelButton[7], val8 := "ProdDataInterfaceHmi".colorCodeLimitSelButton[8], value => "ProdDataInterfaceHmi".colorCodeLimitSummary)   // Limit_ColorCode_Summary: = 2 -> Alarm. Prüfung rechter FB-Aufruf nur, wenn hier KEIN Alarm (VALUE = 0) ansteht; Alarm ist höher prior. / Limit value = 2 -> Alarm. Limit_ColorCode_Summary := 2. Call right block only, if NO alarm (VALUE = 0) is pending here; alarm is higher prior.
      { S7_Templates := "SrcType := UInt" } EQ_Contact(in1 := "ProdDataInterfaceHmi".colorCodeLimitSummary, in2 := 0)
      "InstCompValEqOr2"(compareValue := 1, val1 := "ProdDataInterfaceHmi".colorCodeLimitSelButton[1], val2 := "ProdDataInterfaceHmi".colorCodeLimitSelButton[2], val3 := "ProdDataInterfaceHmi".colorCodeLimitSelButton[3], val4 := "ProdDataInterfaceHmi".colorCodeLimitSelButton[4], val5 := "ProdDataInterfaceHmi".colorCodeLimitSelButton[5], val6 := "ProdDataInterfaceHmi".colorCodeLimitSelButton[6], val7 := "ProdDataInterfaceHmi".colorCodeLimitSelButton[7], val8 := "ProdDataInterfaceHmi".colorCodeLimitSelButton[8], value => "ProdDataInterfaceHmi".colorCodeLimitSummary)   // Grenzwert hat Vorwarngrenze erreicht. Limit_ColorCode_Summary := 1. / Limit value <= Prewarn value. Limit_ColorCode_Summary := 1.
   END_RUNG
   // the same network as SCL:
   "InstLimitValueDataset1"(numberConfigDataSets := "NO_DATASETS_LIMITVALUES",   // "LSicar_ProdDataLimitValues"
                           dataSetNumber := 1,
                           numberOfDataSets := "ProdDataInterfaceHmi".numberOfDataSets,
                           dataSet := "ProdDataInterfaceHmi".limitDataSet[1],
                           colorCodeSelectButton := "ProdDataInterfaceHmi".colorCodeLimitSelButton[1]);
   "InstLimitValueDataset2"(numberConfigDataSets := "NO_DATASETS_LIMITVALUES",   // "LSicar_ProdDataLimitValues"
                           dataSetNumber := 2,
                           numberOfDataSets := "ProdDataInterfaceHmi".numberOfDataSets,
                           dataSet := "ProdDataInterfaceHmi".limitDataSet[2],
                           colorCodeSelectButton := "ProdDataInterfaceHmi".colorCodeLimitSelButton[2]);
   "ProdDataInterfaceHmi".limitDataSet[1].userInterfaceVisibility := "ProdDataSimulation".ProdDataLimitValues.userInterfaceVisibilityDataSet1LimitValues;
   "ProdDataInterfaceHmi".limitDataSet[2].userInterfaceVisibility := "ProdDataSimulation".ProdDataLimitValues.userInterfaceVisibilityDataSet2LimitValues;
   "InstCompValEqOr1"(compareValue := 2,   // "CompValEqOr": Limit_ColorCode_Summary: = 2 -> Alarm. Prüfung rechter FB-Aufruf nur, wenn hier KEIN Alarm (VALUE = 0) ansteht; Alarm ist höher prior. / Limit value = 2 -> Alarm. Limit_ColorCode_Summary := 2. Call right block only, if NO alarm (VALUE = 0) is pending here; alarm is higher prior.
                      val1 := "ProdDataInterfaceHmi".colorCodeLimitSelButton[1],
                      val2 := "ProdDataInterfaceHmi".colorCodeLimitSelButton[2],
                      val3 := "ProdDataInterfaceHmi".colorCodeLimitSelButton[3],
                      val4 := "ProdDataInterfaceHmi".colorCodeLimitSelButton[4],
                      val5 := "ProdDataInterfaceHmi".colorCodeLimitSelButton[5],
                      val6 := "ProdDataInterfaceHmi".colorCodeLimitSelButton[6],
                      val7 := "ProdDataInterfaceHmi".colorCodeLimitSelButton[7],
                      val8 := "ProdDataInterfaceHmi".colorCodeLimitSelButton[8],
                      value => "ProdDataInterfaceHmi".colorCodeLimitSummary,
                      ENO => #_w1);
   IF #_w1 AND ("ProdDataInterfaceHmi".colorCodeLimitSummary = 0) THEN
       "InstCompValEqOr2"(compareValue := 1,   // "CompValEqOr": Grenzwert hat Vorwarngrenze erreicht. Limit_ColorCode_Summary := 1. / Limit value <= Prewarn value. Limit_ColorCode_Summary := 1.
                          val1 := "ProdDataInterfaceHmi".colorCodeLimitSelButton[1],
                          val2 := "ProdDataInterfaceHmi".colorCodeLimitSelButton[2],
                          val3 := "ProdDataInterfaceHmi".colorCodeLimitSelButton[3],
                          val4 := "ProdDataInterfaceHmi".colorCodeLimitSelButton[4],
                          val5 := "ProdDataInterfaceHmi".colorCodeLimitSelButton[5],
                          val6 := "ProdDataInterfaceHmi".colorCodeLimitSelButton[6],
                          val7 := "ProdDataInterfaceHmi".colorCodeLimitSelButton[7],
                          val8 := "ProdDataInterfaceHmi".colorCodeLimitSelButton[8],
                          value => "ProdDataInterfaceHmi".colorCodeLimitSummary);
   END_IF;
END_REGION

REGION Network 7: Beispiel: Shift Counter 1..2 / Call production data shift counter
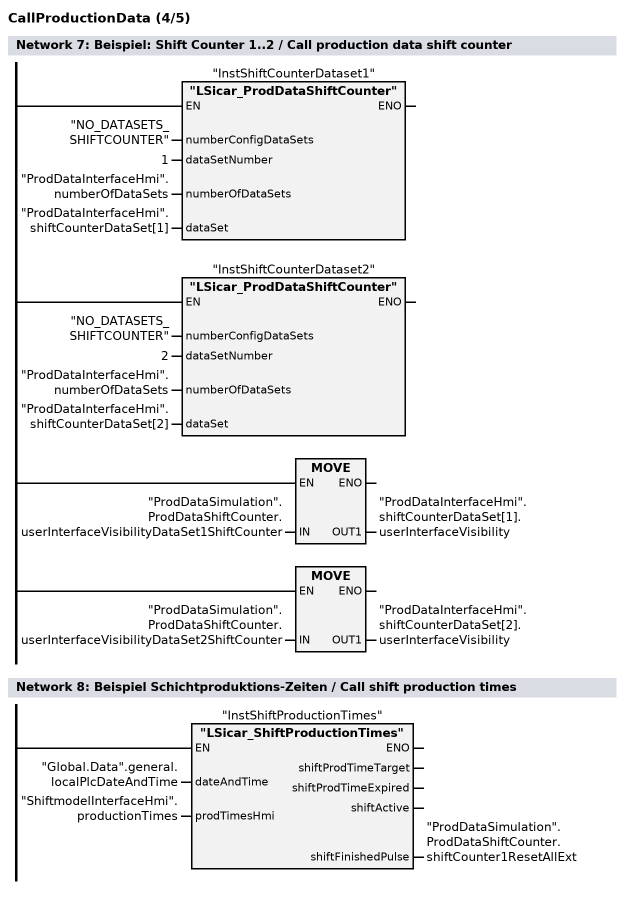
   RUNG wire#powerrail
      "InstShiftCounterDataset1"(numberConfigDataSets := "NO_DATASETS_SHIFTCOUNTER", dataSetNumber := 1, numberOfDataSets := "ProdDataInterfaceHmi".numberOfDataSets, dataSet := "ProdDataInterfaceHmi".shiftCounterDataSet[1])
   END_RUNG
   RUNG wire#powerrail
      "InstShiftCounterDataset2"(numberConfigDataSets := "NO_DATASETS_SHIFTCOUNTER", dataSetNumber := 2, numberOfDataSets := "ProdDataInterfaceHmi".numberOfDataSets, dataSet := "ProdDataInterfaceHmi".shiftCounterDataSet[2])
   END_RUNG
   RUNG wire#powerrail
      Move(in := "ProdDataSimulation".ProdDataShiftCounter.userInterfaceVisibilityDataSet1ShiftCounter, out1 => "ProdDataInterfaceHmi".shiftCounterDataSet[1].userInterfaceVisibility)
   END_RUNG
   RUNG wire#powerrail
      Move(in := "ProdDataSimulation".ProdDataShiftCounter.userInterfaceVisibilityDataSet2ShiftCounter, out1 => "ProdDataInterfaceHmi".shiftCounterDataSet[2].userInterfaceVisibility)
   END_RUNG
   // the same network as SCL:
   "InstShiftCounterDataset1"(numberConfigDataSets := "NO_DATASETS_SHIFTCOUNTER",   // "LSicar_ProdDataShiftCounter"
                           dataSetNumber := 1,
                           numberOfDataSets := "ProdDataInterfaceHmi".numberOfDataSets,
                           dataSet := "ProdDataInterfaceHmi".shiftCounterDataSet[1]);
   "InstShiftCounterDataset2"(numberConfigDataSets := "NO_DATASETS_SHIFTCOUNTER",   // "LSicar_ProdDataShiftCounter"
                           dataSetNumber := 2,
                           numberOfDataSets := "ProdDataInterfaceHmi".numberOfDataSets,
                           dataSet := "ProdDataInterfaceHmi".shiftCounterDataSet[2]);
   "ProdDataInterfaceHmi".shiftCounterDataSet[1].userInterfaceVisibility := "ProdDataSimulation".ProdDataShiftCounter.userInterfaceVisibilityDataSet1ShiftCounter;
   "ProdDataInterfaceHmi".shiftCounterDataSet[2].userInterfaceVisibility := "ProdDataSimulation".ProdDataShiftCounter.userInterfaceVisibilityDataSet2ShiftCounter;
END_REGION

REGION Network 8: Beispiel Schichtproduktions-Zeiten / Call shift production times
   RUNG wire#powerrail
      "InstShiftProductionTimes"(dateAndTime := "Global.Data".general.localPlcDateAndTime, prodTimesHmi := "ShiftmodelInterfaceHmi".productionTimes, shiftProdTimeTarget =>, shiftProdTimeExpired =>, shiftActive =>, shiftFinishedPulse => "ProdDataSimulation".ProdDataShiftCounter.shiftCounter1ResetAllExt)
   END_RUNG
   // the same network as SCL:
   "InstShiftProductionTimes"(dateAndTime := "Global.Data".general.localPlcDateAndTime,   // "LSicar_ShiftProductionTimes"
                           prodTimesHmi := "ShiftmodelInterfaceHmi".productionTimes,
                           shiftFinishedPulse => "ProdDataSimulation".ProdDataShiftCounter.shiftCounter1ResetAllExt);
END_REGION

REGION Network 9: Beispiel: Shift Counter 1..2 + OEE + Trend / Call production data shift counter OEE
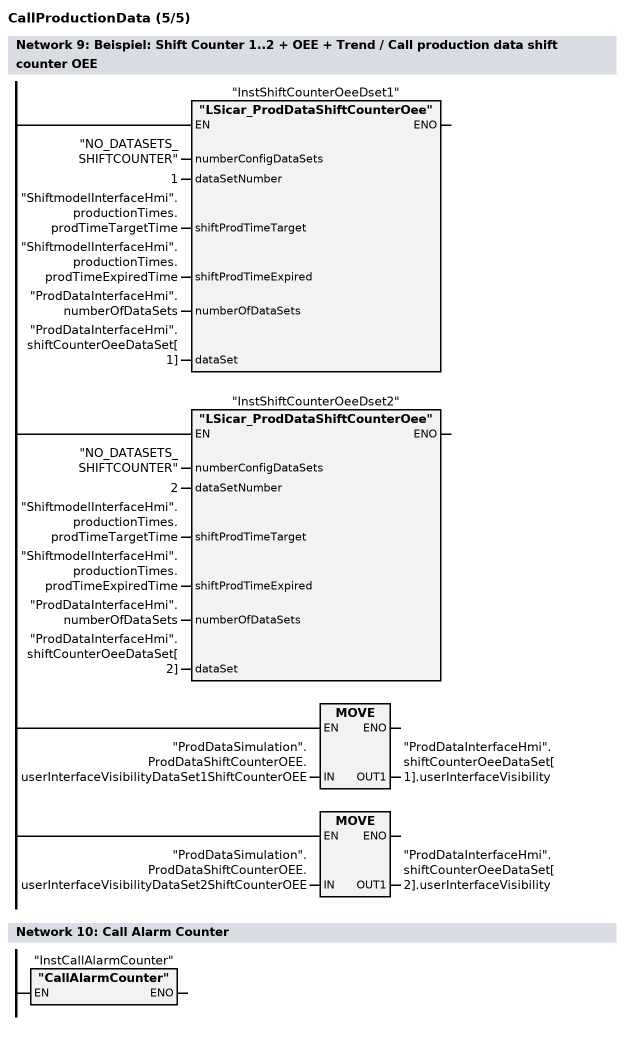
   RUNG wire#powerrail
      "InstShiftCounterOeeDset1"(numberConfigDataSets := "NO_DATASETS_SHIFTCOUNTER", dataSetNumber := 1, shiftProdTimeTarget := "ShiftmodelInterfaceHmi".productionTimes.prodTimeTargetTime, shiftProdTimeExpired := "ShiftmodelInterfaceHmi".productionTimes.prodTimeExpiredTime, numberOfDataSets := "ProdDataInterfaceHmi".numberOfDataSets, dataSet := "ProdDataInterfaceHmi".shiftCounterOeeDataSet[1])
   END_RUNG
   RUNG wire#powerrail
      "InstShiftCounterOeeDset2"(numberConfigDataSets := "NO_DATASETS_SHIFTCOUNTER", dataSetNumber := 2, shiftProdTimeTarget := "ShiftmodelInterfaceHmi".productionTimes.prodTimeTargetTime, shiftProdTimeExpired := "ShiftmodelInterfaceHmi".productionTimes.prodTimeExpiredTime, numberOfDataSets := "ProdDataInterfaceHmi".numberOfDataSets, dataSet := "ProdDataInterfaceHmi".shiftCounterOeeDataSet[2])
   END_RUNG
   RUNG wire#powerrail
      Move(in := "ProdDataSimulation".ProdDataShiftCounterOEE.userInterfaceVisibilityDataSet1ShiftCounterOEE, out1 => "ProdDataInterfaceHmi".shiftCounterOeeDataSet[1].userInterfaceVisibility)
   END_RUNG
   RUNG wire#powerrail
      Move(in := "ProdDataSimulation".ProdDataShiftCounterOEE.userInterfaceVisibilityDataSet2ShiftCounterOEE, out1 => "ProdDataInterfaceHmi".shiftCounterOeeDataSet[2].userInterfaceVisibility)
   END_RUNG
   // the same network as SCL:
   "InstShiftCounterOeeDset1"(numberConfigDataSets := "NO_DATASETS_SHIFTCOUNTER",   // "LSicar_ProdDataShiftCounterOee"
                           dataSetNumber := 1,
                           shiftProdTimeTarget := "ShiftmodelInterfaceHmi".productionTimes.prodTimeTargetTime,
                           shiftProdTimeExpired := "ShiftmodelInterfaceHmi".productionTimes.prodTimeExpiredTime,
                           numberOfDataSets := "ProdDataInterfaceHmi".numberOfDataSets,
                           dataSet := "ProdDataInterfaceHmi".shiftCounterOeeDataSet[1]);
   "InstShiftCounterOeeDset2"(numberConfigDataSets := "NO_DATASETS_SHIFTCOUNTER",   // "LSicar_ProdDataShiftCounterOee"
                           dataSetNumber := 2,
                           shiftProdTimeTarget := "ShiftmodelInterfaceHmi".productionTimes.prodTimeTargetTime,
                           shiftProdTimeExpired := "ShiftmodelInterfaceHmi".productionTimes.prodTimeExpiredTime,
                           numberOfDataSets := "ProdDataInterfaceHmi".numberOfDataSets,
                           dataSet := "ProdDataInterfaceHmi".shiftCounterOeeDataSet[2]);
   "ProdDataInterfaceHmi".shiftCounterOeeDataSet[1].userInterfaceVisibility := "ProdDataSimulation".ProdDataShiftCounterOEE.userInterfaceVisibilityDataSet1ShiftCounterOEE;
   "ProdDataInterfaceHmi".shiftCounterOeeDataSet[2].userInterfaceVisibility := "ProdDataSimulation".ProdDataShiftCounterOEE.userInterfaceVisibilityDataSet2ShiftCounterOEE;
END_REGION

REGION Network 10: Call Alarm Counter
   RUNG wire#powerrail
      "InstCallAlarmCounter"()
   END_RUNG
   // the same network as SCL:
   "InstCallAlarmCounter"();   // "CallAlarmCounter"
END_REGION
END_FUNCTION

FUNCTION "ProductDataSimulation" : Void
{ S7_Optimized_Access := 'TRUE' ; Published := 'FALSE' }
VERSION : 0.1
//Block for simulate the Production Counter

BEGIN
	REGION BLOCK INFO HEADER
	    //===============================================================================
	    // Siemens AG / (c)Copyright 2023
	    //-------------------------------------------------------------------------------
	    // Title:            ProductDataSimulation (FC 4)
	    // Comment/Function: Block for simulate the Production Counter
	    // Library/Family:   Automation Framework
	    // Author:           -
	    // Tested with:      -
	    // Engineering:      TIA Portal V19
	    // Restrictions:     -
	    // Requirements:     -
	    //-------------------------------------------------------------------------------
	    // Change log table:
	    // Version  | Date       | Expert in charge              | Changes applied
	    //----------|------------|-------------------------------|-----------------------------
	    // 01.00.00 | 11.12.2023 |Siemens Industry Online Support| First released version
	    //===============================================================================    
	END_REGION
	
	REGION DESCRIPTION
	   (/*
	 This module is used to simulate the Production Counter:
	*  ProdDataCounter
	*  ProdDataCycleTimer
	*  ProdDataLimitValues
	*  ProdDataShiftCounter
	*  ProdDataShiftCounterOEE
	    
	The data in the data block ("ProdDataSimulation_ProdData") are written to the parameters in The "ProdDataInterfaceHmi".
	This allows the visual representation of the counters be displayed
	*/) 
	    
	    
	END_REGION
	REGION ProdDataCounter
	
	    // Implement an example counter for PrdDataCounter 1 and ProdDataCounter 2
	    IF "ProdDataSimulation".ProdDataCounter.ProdDataEnable THEN
	        
	        // ProdDataCounter 1
	        "ProdDataInterfaceHmi".counterDataSet[1].control[1].countUp := "ProdDataSimulation".ProdDataCounter.ProdDataCounter1Up1;
	        "ProdDataInterfaceHmi".counterDataSet[1].control[1].countDown := "ProdDataSimulation".ProdDataCounter.ProdDataCounter1Down1;
	        "ProdDataInterfaceHmi".counterDataSet[1].control[2].countUp := "ProdDataSimulation".ProdDataCounter.ProdDataCounter1Up2;
	        "ProdDataInterfaceHmi".counterDataSet[1].control[2].countDown := "ProdDataSimulation".ProdDataCounter.ProdDataCounter1Down2;
	        "ProdDataInterfaceHmi".counterDataSet[1].control[1].reset := "ProdDataSimulation".ProdDataCounter.ProdDataCounter1Reset1;
	        "ProdDataInterfaceHmi".counterDataSet[1].control[2].reset := "ProdDataSimulation".ProdDataCounter.ProdDataCounter1Reset2;
	        "ProdDataInterfaceHmi".counterDataSet[1].resetAllExt := "ProdDataSimulation".ProdDataCounter.ProdDataCounter1ResetAll;
	        
	        // ProdDataCounter 2
	        "ProdDataInterfaceHmi".counterDataSet[2].control[1].countUp := "ProdDataSimulation".ProdDataCounter.ProdDataCounter2Up1;
	        "ProdDataInterfaceHmi".counterDataSet[2].control[1].countDown := "ProdDataSimulation".ProdDataCounter.ProdDataCounter2Down1;
	        "ProdDataInterfaceHmi".counterDataSet[2].control[2].countUp := "ProdDataSimulation".ProdDataCounter.ProdDataCounter2Up2;
	        "ProdDataInterfaceHmi".counterDataSet[2].control[2].countDown := "ProdDataSimulation".ProdDataCounter.ProdDataCounter2Down2;
	        "ProdDataInterfaceHmi".counterDataSet[2].control[1].reset := "ProdDataSimulation".ProdDataCounter.ProdDataCounter2Reset1;
	        "ProdDataInterfaceHmi".counterDataSet[2].control[2].reset := "ProdDataSimulation".ProdDataCounter.ProdDataCounter2Reset2;
	        "ProdDataInterfaceHmi".counterDataSet[2].resetAllExt := "ProdDataSimulation".ProdDataCounter.ProdDataCounter2ResetAll;
	        
	        //Via the user interface „.userInterfaceVisibility“ [DWord] individual values can be hidden in the visualization
	        "ProdDataInterfaceHmi".counterDataSet[1].userInterfaceVisibility := "ProdDataSimulation".ProdDataCounter.userInterfaceVisibilityDataSet1Counter;
	        "ProdDataInterfaceHmi".counterDataSet[2].userInterfaceVisibility := "ProdDataSimulation".ProdDataCounter.userInterfaceVisibilityDataSet2Counter;
	    END_IF;
	    
	END_REGION
	
	REGION CycleTimer
	    // Example to demonstrate and test the functionality of the cycle timer
	    IF "ProdDataSimulation".ProdDataCyclic.cyclicTimerEnable THEN
	        
	        "ProdDataInterfaceHmi".cycleTimerDataSet[1].control[1].run := "ProdDataSimulation".ProdDataCyclic.cycleTimer1Run1;
	        "ProdDataInterfaceHmi".cycleTimerDataSet[1].control[1].hold := "ProdDataSimulation".ProdDataCyclic.cycleTimer1Hold1;
	        "ProdDataInterfaceHmi".cycleTimerDataSet[1].control[1].reset := "ProdDataSimulation".ProdDataCyclic.cycleTimer1Reset1;
	        "ProdDataInterfaceHmi".cycleTimerDataSet[1].control[2].run := "ProdDataSimulation".ProdDataCyclic.cycleTimer1Run2;
	        "ProdDataInterfaceHmi".cycleTimerDataSet[1].control[2].hold := "ProdDataSimulation".ProdDataCyclic.cycleTimer1Hold2;
	        "ProdDataInterfaceHmi".cycleTimerDataSet[1].control[2].reset := "ProdDataSimulation".ProdDataCyclic.cycleTimer1Reset2;
	        "ProdDataInterfaceHmi".cycleTimerDataSet[2].control[1].run := "ProdDataSimulation".ProdDataCyclic.cycleTimer2Run1;
	        "ProdDataInterfaceHmi".cycleTimerDataSet[2].control[1].hold := "ProdDataSimulation".ProdDataCyclic.cycleTimer2Hold1;
	        "ProdDataInterfaceHmi".cycleTimerDataSet[2].control[1].reset := "ProdDataSimulation".ProdDataCyclic.cycleTimer2Reset1;
	        "ProdDataInterfaceHmi".cycleTimerDataSet[2].control[2].run := "ProdDataSimulation".ProdDataCyclic.cycleTimer2Run2;
	        "ProdDataInterfaceHmi".cycleTimerDataSet[2].control[2].hold := "ProdDataSimulation".ProdDataCyclic.cycleTimer2Hold2;
	        "ProdDataInterfaceHmi".cycleTimerDataSet[2].control[2].reset := "ProdDataSimulation".ProdDataCyclic.cycleTimer2Reset2;
	        "ProdDataInterfaceHmi".cycleTimerDataSet[1].resetAverageAllExt := "ProdDataSimulation".ProdDataCyclic.cycleTimer1ResetAll;
	        "ProdDataInterfaceHmi".cycleTimerDataSet[2].resetAverageAllExt := "ProdDataSimulation".ProdDataCyclic.cycleTimer2ResetAll;
	        
	        //Via the user interface „.userInterfaceVisibility“ [DWord] individual values can be hidden in the visualization
	        "ProdDataInterfaceHmi".cycleTimerDataSet[1].userInterfaceVisibility := "ProdDataSimulation".ProdDataCyclic.userInterfaceVisibilityDataSet1Cyclic;
	        "ProdDataInterfaceHmi".cycleTimerDataSet[2].userInterfaceVisibility := "ProdDataSimulation".ProdDataCyclic.userInterfaceVisibilityDataSet2Cyclic;
	        
	    END_IF;
	END_REGION
	
	
	REGION LimitValues
	    // Example to demonstrate and test the functionality of the limit counters
	
	    IF "ProdDataSimulation".ProdDataLimitValues.limitValuesEnable THEN
	        
	        "ProdDataInterfaceHmi".limitDataSet[1].control[1].count := "ProdDataSimulation".ProdDataLimitValues.limitVal1Count1;
	        "ProdDataInterfaceHmi".limitDataSet[1].control[1].set := "ProdDataSimulation".ProdDataLimitValues.limitVal1Set1;
	        "ProdDataSimulation".ProdDataLimitValues.limitVal1Count1PreWarn1 := "ProdDataInterfaceHmi".limitDataSet[1].control[1].prewarn;
	        "ProdDataSimulation".ProdDataLimitValues.limitVal1Count1Alarm1 := "ProdDataInterfaceHmi".limitDataSet[1].control[1].alarm;
	        "ProdDataInterfaceHmi".limitDataSet[1].control[2].count := "ProdDataSimulation".ProdDataLimitValues.limitVal1Count2;
	        "ProdDataInterfaceHmi".limitDataSet[1].control[2].set := "ProdDataSimulation".ProdDataLimitValues.limitVal1Set2;
	        "ProdDataSimulation".ProdDataLimitValues.limitVal1Count1PreWarn2 := "ProdDataInterfaceHmi".limitDataSet[1].control[2].prewarn;
	        "ProdDataSimulation".ProdDataLimitValues.limitVal1Count1Alarm2 := "ProdDataInterfaceHmi".limitDataSet[1].control[2].alarm;
	        "ProdDataInterfaceHmi".limitDataSet[1].control[3].count := "ProdDataSimulation".ProdDataLimitValues.limitVal1Count3;
	        "ProdDataInterfaceHmi".limitDataSet[1].control[3].set := "ProdDataSimulation".ProdDataLimitValues.limitVal1Set3;
	        "ProdDataSimulation".ProdDataLimitValues.limitVal1Count1PreWarn3 := "ProdDataInterfaceHmi".limitDataSet[1].control[3].prewarn;
	        "ProdDataSimulation".ProdDataLimitValues.limitVal1Count1Alarm3 := "ProdDataInterfaceHmi".limitDataSet[1].control[3].alarm;
	        
	        //Via the user interface „.userInterfaceVisibility“ [DWord] individual values can be hidden in the visualization
	        "ProdDataInterfaceHmi".limitDataSet[1].userInterfaceVisibility := "ProdDataSimulation".ProdDataLimitValues.userInterfaceVisibilityDataSet1LimitValues;
	        "ProdDataInterfaceHmi".limitDataSet[2].userInterfaceVisibility := "ProdDataSimulation".ProdDataLimitValues.userInterfaceVisibilityDataSet2LimitValues;
	    END_IF;
	END_REGION
	
	REGION ShiftCounter
	    //Example to demonstrate and test the functionality of the shift counters
	    IF "ProdDataSimulation".ProdDataShiftCounter.ShiftCounterEnable THEN
	        
	        "ProdDataInterfaceHmi".shiftCounterDataSet[1].countPartsCurrent[1] := "ProdDataSimulation".ProdDataShiftCounter.shiftCounter1Cnt1Curr;
	        "ProdDataInterfaceHmi".shiftCounterDataSet[1].countPartsCurrent[2] := "ProdDataSimulation".ProdDataShiftCounter.shiftCounter1Cnt2Curr;
	        "ProdDataInterfaceHmi".shiftCounterDataSet[1].countPartsCurrent[3] := "ProdDataSimulation".ProdDataShiftCounter.shiftCounter1Cnt3Curr;
	        "ProdDataInterfaceHmi".shiftCounterDataSet[1].resetAllExt := "ProdDataSimulation".ProdDataShiftCounter.shiftCounter1ResetAllExt;
	        
	     //Via the user interface „.userInterfaceVisibility“ [DWord] individual values can be hidden in the visualization
	        "ProdDataInterfaceHmi".shiftCounterDataSet[1].userInterfaceVisibility := "ProdDataSimulation".ProdDataShiftCounter.userInterfaceVisibilityDataSet1ShiftCounter;
	        "ProdDataInterfaceHmi".shiftCounterDataSet[2].userInterfaceVisibility := "ProdDataSimulation".ProdDataShiftCounter.userInterfaceVisibilityDataSet2ShiftCounter;
	    END_IF;
	    
	END_REGION
	
	REGION ShiftCounterOEE
	    // Example to demonstrate and test the functionality of the shift counter OEE
	    
	    IF "ProdDataSimulation".ProdDataShiftCounterOEE.ShiftCounterOEEEnable THEN
	        
	        "ProdDataInterfaceHmi".shiftCounterOeeDataSet[1].countPartsCurrent[1] := "ProdDataSimulation".ProdDataShiftCounter.shiftCounter1Cnt1Curr;
	        "ProdDataInterfaceHmi".shiftCounterOeeDataSet[1].countPartsCurrent[2] := "ProdDataSimulation".ProdDataShiftCounter.shiftCounter1Cnt2Curr;
	        "ProdDataInterfaceHmi".shiftCounterOeeDataSet[1].countPartsCurrent[3] := "ProdDataSimulation".ProdDataShiftCounter.shiftCounter1Cnt3Curr;
	        "ProdDataInterfaceHmi".shiftCounterOeeDataSet[1].countPartsCurrentOk[1] := "ProdDataSimulation".ProdDataShiftCounter.shiftCounter1Cnt1CurrOk;
	        "ProdDataInterfaceHmi".shiftCounterOeeDataSet[1].countPartsCurrentOk[2] := "ProdDataSimulation".ProdDataShiftCounter.shiftCounter1Cnt2CurrOk;
	        "ProdDataInterfaceHmi".shiftCounterOeeDataSet[1].countPartsCurrentOk[3] := "ProdDataSimulation".ProdDataShiftCounter.shiftCounter1Cnt3CurrOk;
	        
	     //Via the user interface „.userInterfaceVisibility“ [DWord] individual values can be hidden in the visualization
	        "ProdDataInterfaceHmi".shiftCounterOeeDataSet[1].userInterfaceVisibility := "ProdDataSimulation".ProdDataShiftCounterOEE.userInterfaceVisibilityDataSet1ShiftCounterOEE;
	        "ProdDataInterfaceHmi".shiftCounterOeeDataSet[2].userInterfaceVisibility := "ProdDataSimulation".ProdDataShiftCounterOEE.userInterfaceVisibilityDataSet2ShiftCounterOEE;
	    END_IF;
	END_REGION
	
	
	
END_FUNCTION

FUNCTION_BLOCK "CallProcessCount"   // FB2, LAD
// stored: MemoryReserve 100, SetENOAutomatically false
   VAR
      statPulse { ExternalAccessible := 'False'; ExternalVisible := 'False'; ExternalWritable := 'False'} : Array[0..299] of Bool;
   END_VAR
   VAR_TEMP
      tempEnter : Bool;   // Enter the conditions for the count to increase.
   END_VAR
   VAR_TEMP   // added for the SCL form of the ladder/FBD networks
      _w1 : Bool;
   END_VAR
BEGIN

REGION Network 1: Production Data 1 Anode NG Parts
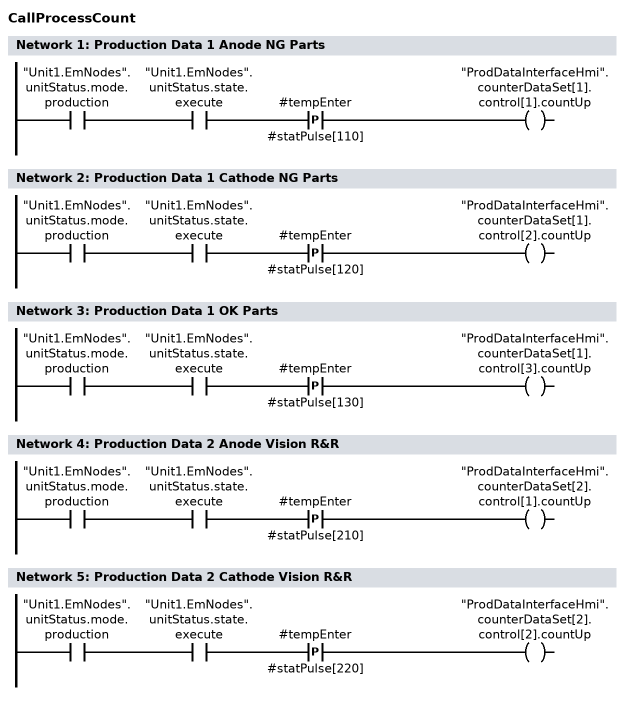
   RUNG wire#powerrail
      Contact( "Unit1.EmNodes".unitStatus.mode.production )
      Contact( "Unit1.EmNodes".unitStatus.state.execute )
      P_Contact(operand := #tempEnter, bit := #statPulse[110])
      Coil( "ProdDataInterfaceHmi".counterDataSet[1].control[1].countUp )
   END_RUNG
   // the same network as SCL:
   #_w1 := "Unit1.EmNodes".unitStatus.mode.production AND "Unit1.EmNodes".unitStatus.state.execute AND #tempEnter AND NOT #statPulse[110];   // rising edge of #tempEnter
   #statPulse[110] := #tempEnter;
   "ProdDataInterfaceHmi".counterDataSet[1].control[1].countUp := #_w1;
END_REGION

REGION Network 2: Production Data 1 Cathode NG Parts
   RUNG wire#powerrail
      Contact( "Unit1.EmNodes".unitStatus.mode.production )
      Contact( "Unit1.EmNodes".unitStatus.state.execute )
      P_Contact(operand := #tempEnter, bit := #statPulse[120])
      Coil( "ProdDataInterfaceHmi".counterDataSet[1].control[2].countUp )
   END_RUNG
   // the same network as SCL:
   #_w1 := "Unit1.EmNodes".unitStatus.mode.production AND "Unit1.EmNodes".unitStatus.state.execute AND #tempEnter AND NOT #statPulse[120];   // rising edge of #tempEnter
   #statPulse[120] := #tempEnter;
   "ProdDataInterfaceHmi".counterDataSet[1].control[2].countUp := #_w1;
END_REGION

REGION Network 3: Production Data 1 OK Parts
   RUNG wire#powerrail
      Contact( "Unit1.EmNodes".unitStatus.mode.production )
      Contact( "Unit1.EmNodes".unitStatus.state.execute )
      P_Contact(operand := #tempEnter, bit := #statPulse[130])
      Coil( "ProdDataInterfaceHmi".counterDataSet[1].control[3].countUp )
   END_RUNG
   // the same network as SCL:
   #_w1 := "Unit1.EmNodes".unitStatus.mode.production AND "Unit1.EmNodes".unitStatus.state.execute AND #tempEnter AND NOT #statPulse[130];   // rising edge of #tempEnter
   #statPulse[130] := #tempEnter;
   "ProdDataInterfaceHmi".counterDataSet[1].control[3].countUp := #_w1;
END_REGION

REGION Network 4: Production Data 2 Anode Vision R&R
   RUNG wire#powerrail
      Contact( "Unit1.EmNodes".unitStatus.mode.production )
      Contact( "Unit1.EmNodes".unitStatus.state.execute )
      P_Contact(operand := #tempEnter, bit := #statPulse[210])
      Coil( "ProdDataInterfaceHmi".counterDataSet[2].control[1].countUp )
   END_RUNG
   // the same network as SCL:
   #_w1 := "Unit1.EmNodes".unitStatus.mode.production AND "Unit1.EmNodes".unitStatus.state.execute AND #tempEnter AND NOT #statPulse[210];   // rising edge of #tempEnter
   #statPulse[210] := #tempEnter;
   "ProdDataInterfaceHmi".counterDataSet[2].control[1].countUp := #_w1;
END_REGION

REGION Network 5: Production Data 2 Cathode Vision R&R
   RUNG wire#powerrail
      Contact( "Unit1.EmNodes".unitStatus.mode.production )
      Contact( "Unit1.EmNodes".unitStatus.state.execute )
      P_Contact(operand := #tempEnter, bit := #statPulse[220])
      Coil( "ProdDataInterfaceHmi".counterDataSet[2].control[2].countUp )
   END_RUNG
   // the same network as SCL:
   #_w1 := "Unit1.EmNodes".unitStatus.mode.production AND "Unit1.EmNodes".unitStatus.state.execute AND #tempEnter AND NOT #statPulse[220];   // rising edge of #tempEnter
   #statPulse[220] := #tempEnter;
   "ProdDataInterfaceHmi".counterDataSet[2].control[2].countUp := #_w1;
END_REGION
END_FUNCTION_BLOCK

FUNCTION "CallCycleTimer" : Void   // FC18, LAD
// stored: SetENOAutomatically false
   VAR CONSTANT
      TRUE : Bool := TRUE;
   END_VAR
BEGIN

REGION Network 1: Cycle Timer Em 0
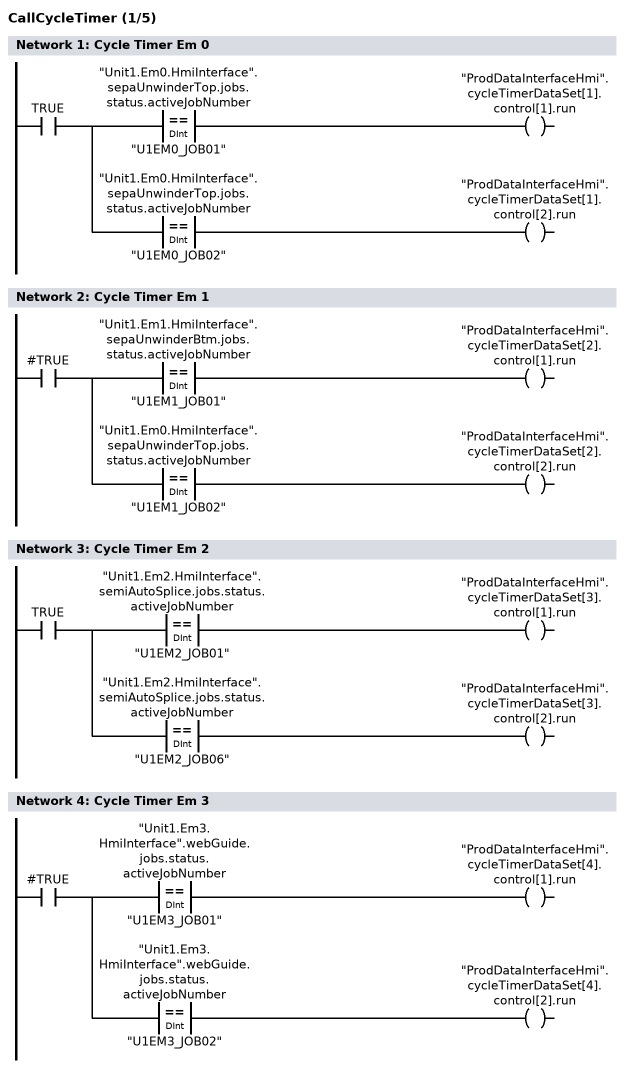
   RUNG wire#powerrail
      Contact( TRUE )
      wire#w1
      { S7_Templates := "SrcType := DInt" } EQ_Contact(in1 := "Unit1.Em0.HmiInterface".sepaUnwinderTop.jobs.status.activeJobNumber, in2 := "U1EM0_JOB01")
      Coil( "ProdDataInterfaceHmi".cycleTimerDataSet[1].control[1].run )
   END_RUNG
   RUNG wire#w1
      { S7_Templates := "SrcType := DInt" } EQ_Contact(in1 := "Unit1.Em0.HmiInterface".sepaUnwinderTop.jobs.status.activeJobNumber, in2 := "U1EM0_JOB02")
      Coil( "ProdDataInterfaceHmi".cycleTimerDataSet[1].control[2].run )
   END_RUNG
   // the same network as SCL:
   "ProdDataInterfaceHmi".cycleTimerDataSet[1].control[1].run := TRUE AND ("Unit1.Em0.HmiInterface".sepaUnwinderTop.jobs.status.activeJobNumber = "U1EM0_JOB01");
   "ProdDataInterfaceHmi".cycleTimerDataSet[1].control[2].run := TRUE AND ("Unit1.Em0.HmiInterface".sepaUnwinderTop.jobs.status.activeJobNumber = "U1EM0_JOB02");
END_REGION

REGION Network 2: Cycle Timer Em 1
   RUNG wire#powerrail
      Contact( #TRUE )
      wire#w1
      { S7_Templates := "SrcType := DInt" } EQ_Contact(in1 := "Unit1.Em1.HmiInterface".sepaUnwinderBtm.jobs.status.activeJobNumber, in2 := "U1EM1_JOB01")
      Coil( "ProdDataInterfaceHmi".cycleTimerDataSet[2].control[1].run )
   END_RUNG
   RUNG wire#w1
      { S7_Templates := "SrcType := DInt" } EQ_Contact(in1 := "Unit1.Em0.HmiInterface".sepaUnwinderTop.jobs.status.activeJobNumber, in2 := "U1EM1_JOB02")
      Coil( "ProdDataInterfaceHmi".cycleTimerDataSet[2].control[2].run )
   END_RUNG
   // the same network as SCL:
   "ProdDataInterfaceHmi".cycleTimerDataSet[2].control[1].run := #TRUE AND ("Unit1.Em1.HmiInterface".sepaUnwinderBtm.jobs.status.activeJobNumber = "U1EM1_JOB01");
   "ProdDataInterfaceHmi".cycleTimerDataSet[2].control[2].run := #TRUE AND ("Unit1.Em0.HmiInterface".sepaUnwinderTop.jobs.status.activeJobNumber = "U1EM1_JOB02");
END_REGION

REGION Network 3: Cycle Timer Em 2
   RUNG wire#powerrail
      Contact( TRUE )
      wire#w1
      { S7_Templates := "SrcType := DInt" } EQ_Contact(in1 := "Unit1.Em2.HmiInterface".semiAutoSplice.jobs.status.activeJobNumber, in2 := "U1EM2_JOB01")
      Coil( "ProdDataInterfaceHmi".cycleTimerDataSet[3].control[1].run )
   END_RUNG
   RUNG wire#w1
      { S7_Templates := "SrcType := DInt" } EQ_Contact(in1 := "Unit1.Em2.HmiInterface".semiAutoSplice.jobs.status.activeJobNumber, in2 := "U1EM2_JOB06")
      Coil( "ProdDataInterfaceHmi".cycleTimerDataSet[3].control[2].run )
   END_RUNG
   // the same network as SCL:
   "ProdDataInterfaceHmi".cycleTimerDataSet[3].control[1].run := TRUE AND ("Unit1.Em2.HmiInterface".semiAutoSplice.jobs.status.activeJobNumber = "U1EM2_JOB01");
   "ProdDataInterfaceHmi".cycleTimerDataSet[3].control[2].run := TRUE AND ("Unit1.Em2.HmiInterface".semiAutoSplice.jobs.status.activeJobNumber = "U1EM2_JOB06");
END_REGION

REGION Network 4: Cycle Timer Em 3
   RUNG wire#powerrail
      Contact( #TRUE )
      wire#w1
      { S7_Templates := "SrcType := DInt" } EQ_Contact(in1 := "Unit1.Em3.HmiInterface".webGuide.jobs.status.activeJobNumber, in2 := "U1EM3_JOB01")
      Coil( "ProdDataInterfaceHmi".cycleTimerDataSet[4].control[1].run )
   END_RUNG
   RUNG wire#w1
      { S7_Templates := "SrcType := DInt" } EQ_Contact(in1 := "Unit1.Em3.HmiInterface".webGuide.jobs.status.activeJobNumber, in2 := "U1EM3_JOB02")
      Coil( "ProdDataInterfaceHmi".cycleTimerDataSet[4].control[2].run )
   END_RUNG
   // the same network as SCL:
   "ProdDataInterfaceHmi".cycleTimerDataSet[4].control[1].run := #TRUE AND ("Unit1.Em3.HmiInterface".webGuide.jobs.status.activeJobNumber = "U1EM3_JOB01");
   "ProdDataInterfaceHmi".cycleTimerDataSet[4].control[2].run := #TRUE AND ("Unit1.Em3.HmiInterface".webGuide.jobs.status.activeJobNumber = "U1EM3_JOB02");
END_REGION

REGION Network 5: Cycle Timer Em 4
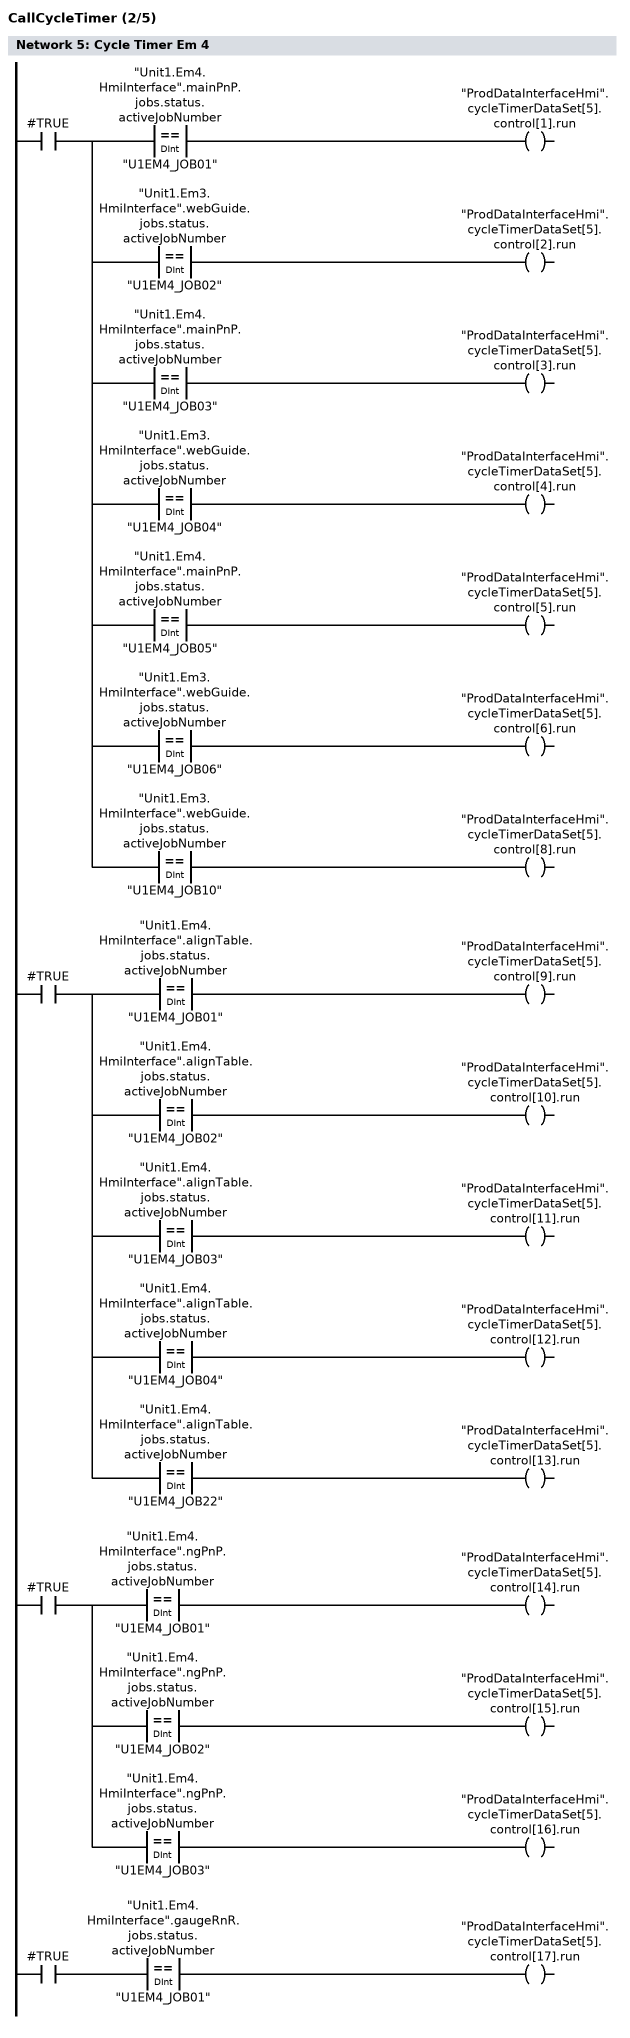
   RUNG wire#powerrail
      Contact( #TRUE )
      wire#w1
      { S7_Templates := "SrcType := DInt" } EQ_Contact(in1 := "Unit1.Em4.HmiInterface".mainPnP.jobs.status.activeJobNumber, in2 := "U1EM4_JOB01")
      Coil( "ProdDataInterfaceHmi".cycleTimerDataSet[5].control[1].run )
   END_RUNG
   RUNG wire#w1
      { S7_Templates := "SrcType := DInt" } EQ_Contact(in1 := "Unit1.Em3.HmiInterface".webGuide.jobs.status.activeJobNumber, in2 := "U1EM4_JOB02")
      Coil( "ProdDataInterfaceHmi".cycleTimerDataSet[5].control[2].run )
   END_RUNG
   RUNG wire#w1
      { S7_Templates := "SrcType := DInt" } EQ_Contact(in1 := "Unit1.Em4.HmiInterface".mainPnP.jobs.status.activeJobNumber, in2 := "U1EM4_JOB03")
      Coil( "ProdDataInterfaceHmi".cycleTimerDataSet[5].control[3].run )
   END_RUNG
   RUNG wire#w1
      { S7_Templates := "SrcType := DInt" } EQ_Contact(in1 := "Unit1.Em3.HmiInterface".webGuide.jobs.status.activeJobNumber, in2 := "U1EM4_JOB04")
      Coil( "ProdDataInterfaceHmi".cycleTimerDataSet[5].control[4].run )
   END_RUNG
   RUNG wire#w1
      { S7_Templates := "SrcType := DInt" } EQ_Contact(in1 := "Unit1.Em4.HmiInterface".mainPnP.jobs.status.activeJobNumber, in2 := "U1EM4_JOB05")
      Coil( "ProdDataInterfaceHmi".cycleTimerDataSet[5].control[5].run )
   END_RUNG
   RUNG wire#w1
      { S7_Templates := "SrcType := DInt" } EQ_Contact(in1 := "Unit1.Em3.HmiInterface".webGuide.jobs.status.activeJobNumber, in2 := "U1EM4_JOB06")
      Coil( "ProdDataInterfaceHmi".cycleTimerDataSet[5].control[6].run )
   END_RUNG
   RUNG wire#w1
      { S7_Templates := "SrcType := DInt" } EQ_Contact(in1 := "Unit1.Em3.HmiInterface".webGuide.jobs.status.activeJobNumber, in2 := "U1EM4_JOB10")
      Coil( "ProdDataInterfaceHmi".cycleTimerDataSet[5].control[8].run )
   END_RUNG
   RUNG wire#powerrail
      Contact( #TRUE )
      wire#w2
      { S7_Templates := "SrcType := DInt" } EQ_Contact(in1 := "Unit1.Em4.HmiInterface".alignTable.jobs.status.activeJobNumber, in2 := "U1EM4_JOB01")
      Coil( "ProdDataInterfaceHmi".cycleTimerDataSet[5].control[9].run )
   END_RUNG
   RUNG wire#w2
      { S7_Templates := "SrcType := DInt" } EQ_Contact(in1 := "Unit1.Em4.HmiInterface".alignTable.jobs.status.activeJobNumber, in2 := "U1EM4_JOB02")
      Coil( "ProdDataInterfaceHmi".cycleTimerDataSet[5].control[10].run )
   END_RUNG
   RUNG wire#w2
      { S7_Templates := "SrcType := DInt" } EQ_Contact(in1 := "Unit1.Em4.HmiInterface".alignTable.jobs.status.activeJobNumber, in2 := "U1EM4_JOB03")
      Coil( "ProdDataInterfaceHmi".cycleTimerDataSet[5].control[11].run )
   END_RUNG
   RUNG wire#w2
      { S7_Templates := "SrcType := DInt" } EQ_Contact(in1 := "Unit1.Em4.HmiInterface".alignTable.jobs.status.activeJobNumber, in2 := "U1EM4_JOB04")
      Coil( "ProdDataInterfaceHmi".cycleTimerDataSet[5].control[12].run )
   END_RUNG
   RUNG wire#w2
      { S7_Templates := "SrcType := DInt" } EQ_Contact(in1 := "Unit1.Em4.HmiInterface".alignTable.jobs.status.activeJobNumber, in2 := "U1EM4_JOB22")
      Coil( "ProdDataInterfaceHmi".cycleTimerDataSet[5].control[13].run )
   END_RUNG
   RUNG wire#powerrail
      Contact( #TRUE )
      wire#w3
      { S7_Templates := "SrcType := DInt" } EQ_Contact(in1 := "Unit1.Em4.HmiInterface".ngPnP.jobs.status.activeJobNumber, in2 := "U1EM4_JOB01")
      Coil( "ProdDataInterfaceHmi".cycleTimerDataSet[5].control[14].run )
   END_RUNG
   RUNG wire#w3
      { S7_Templates := "SrcType := DInt" } EQ_Contact(in1 := "Unit1.Em4.HmiInterface".ngPnP.jobs.status.activeJobNumber, in2 := "U1EM4_JOB02")
      Coil( "ProdDataInterfaceHmi".cycleTimerDataSet[5].control[15].run )
   END_RUNG
   RUNG wire#w3
      { S7_Templates := "SrcType := DInt" } EQ_Contact(in1 := "Unit1.Em4.HmiInterface".ngPnP.jobs.status.activeJobNumber, in2 := "U1EM4_JOB03")
      Coil( "ProdDataInterfaceHmi".cycleTimerDataSet[5].control[16].run )
   END_RUNG
   RUNG wire#powerrail
      Contact( #TRUE )
      { S7_Templates := "SrcType := DInt" } EQ_Contact(in1 := "Unit1.Em4.HmiInterface".gaugeRnR.jobs.status.activeJobNumber, in2 := "U1EM4_JOB01")
      Coil( "ProdDataInterfaceHmi".cycleTimerDataSet[5].control[17].run )
   END_RUNG
   // the same network as SCL:
   "ProdDataInterfaceHmi".cycleTimerDataSet[5].control[1].run := #TRUE AND ("Unit1.Em4.HmiInterface".mainPnP.jobs.status.activeJobNumber = "U1EM4_JOB01");
   "ProdDataInterfaceHmi".cycleTimerDataSet[5].control[2].run := #TRUE AND ("Unit1.Em3.HmiInterface".webGuide.jobs.status.activeJobNumber = "U1EM4_JOB02");
   "ProdDataInterfaceHmi".cycleTimerDataSet[5].control[3].run := #TRUE AND ("Unit1.Em4.HmiInterface".mainPnP.jobs.status.activeJobNumber = "U1EM4_JOB03");
   "ProdDataInterfaceHmi".cycleTimerDataSet[5].control[4].run := #TRUE AND ("Unit1.Em3.HmiInterface".webGuide.jobs.status.activeJobNumber = "U1EM4_JOB04");
   "ProdDataInterfaceHmi".cycleTimerDataSet[5].control[5].run := #TRUE AND ("Unit1.Em4.HmiInterface".mainPnP.jobs.status.activeJobNumber = "U1EM4_JOB05");
   "ProdDataInterfaceHmi".cycleTimerDataSet[5].control[6].run := #TRUE AND ("Unit1.Em3.HmiInterface".webGuide.jobs.status.activeJobNumber = "U1EM4_JOB06");
   "ProdDataInterfaceHmi".cycleTimerDataSet[5].control[8].run := #TRUE AND ("Unit1.Em3.HmiInterface".webGuide.jobs.status.activeJobNumber = "U1EM4_JOB10");
   "ProdDataInterfaceHmi".cycleTimerDataSet[5].control[9].run := #TRUE AND ("Unit1.Em4.HmiInterface".alignTable.jobs.status.activeJobNumber = "U1EM4_JOB01");
   "ProdDataInterfaceHmi".cycleTimerDataSet[5].control[10].run := #TRUE AND ("Unit1.Em4.HmiInterface".alignTable.jobs.status.activeJobNumber = "U1EM4_JOB02");
   "ProdDataInterfaceHmi".cycleTimerDataSet[5].control[11].run := #TRUE AND ("Unit1.Em4.HmiInterface".alignTable.jobs.status.activeJobNumber = "U1EM4_JOB03");
   "ProdDataInterfaceHmi".cycleTimerDataSet[5].control[12].run := #TRUE AND ("Unit1.Em4.HmiInterface".alignTable.jobs.status.activeJobNumber = "U1EM4_JOB04");
   "ProdDataInterfaceHmi".cycleTimerDataSet[5].control[13].run := #TRUE AND ("Unit1.Em4.HmiInterface".alignTable.jobs.status.activeJobNumber = "U1EM4_JOB22");
   "ProdDataInterfaceHmi".cycleTimerDataSet[5].control[14].run := #TRUE AND ("Unit1.Em4.HmiInterface".ngPnP.jobs.status.activeJobNumber = "U1EM4_JOB01");
   "ProdDataInterfaceHmi".cycleTimerDataSet[5].control[15].run := #TRUE AND ("Unit1.Em4.HmiInterface".ngPnP.jobs.status.activeJobNumber = "U1EM4_JOB02");
   "ProdDataInterfaceHmi".cycleTimerDataSet[5].control[16].run := #TRUE AND ("Unit1.Em4.HmiInterface".ngPnP.jobs.status.activeJobNumber = "U1EM4_JOB03");
   "ProdDataInterfaceHmi".cycleTimerDataSet[5].control[17].run := #TRUE AND ("Unit1.Em4.HmiInterface".gaugeRnR.jobs.status.activeJobNumber = "U1EM4_JOB01");
END_REGION

REGION Network 6: Cycle Timer Em 5
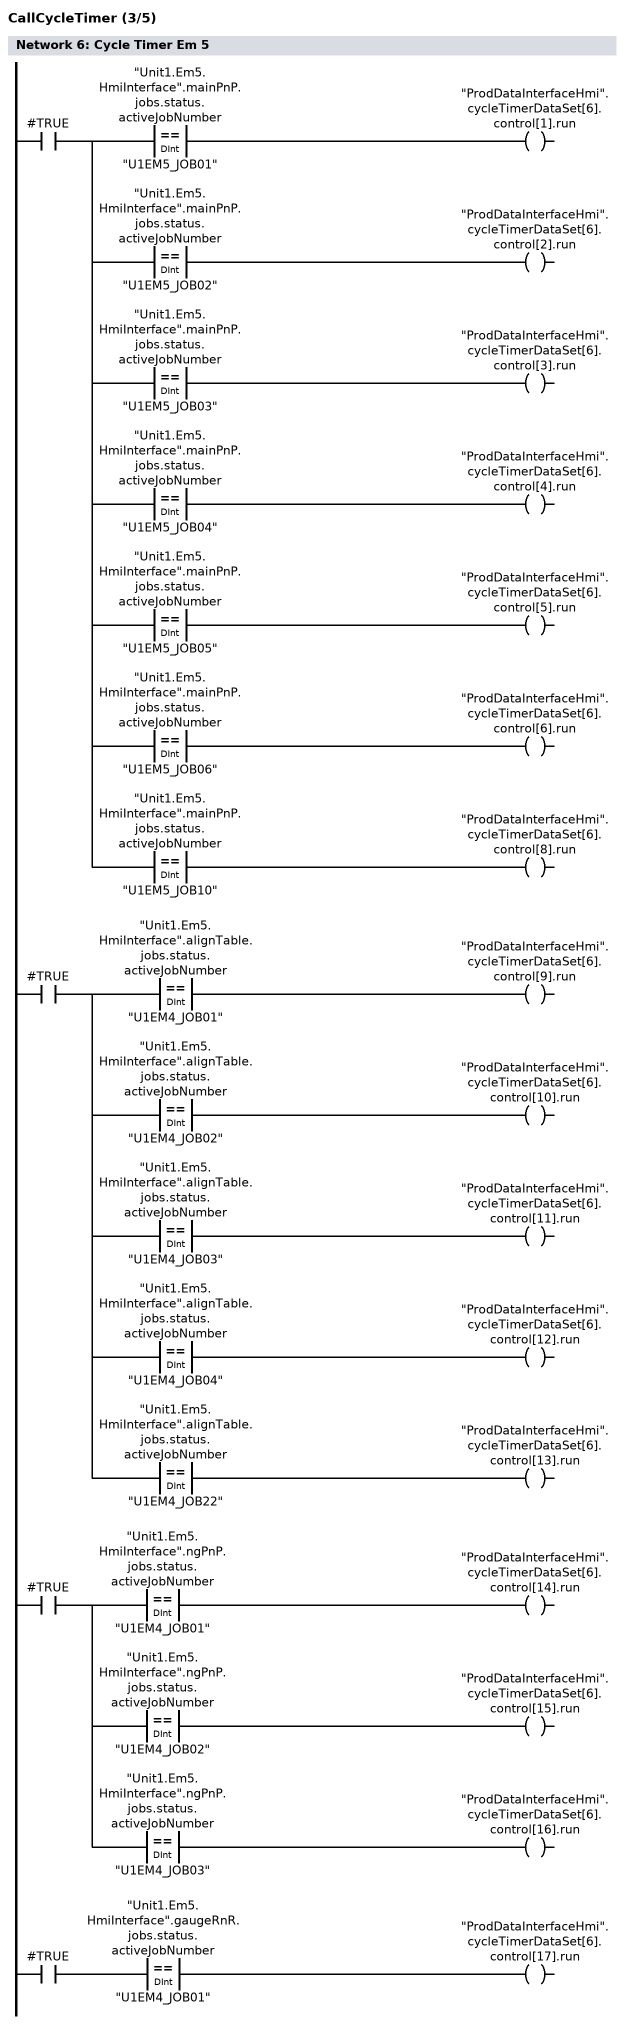
   RUNG wire#powerrail
      Contact( #TRUE )
      wire#w1
      { S7_Templates := "SrcType := DInt" } EQ_Contact(in1 := "Unit1.Em5.HmiInterface".mainPnP.jobs.status.activeJobNumber, in2 := "U1EM5_JOB01")
      Coil( "ProdDataInterfaceHmi".cycleTimerDataSet[6].control[1].run )
   END_RUNG
   RUNG wire#w1
      { S7_Templates := "SrcType := DInt" } EQ_Contact(in1 := "Unit1.Em5.HmiInterface".mainPnP.jobs.status.activeJobNumber, in2 := "U1EM5_JOB02")
      Coil( "ProdDataInterfaceHmi".cycleTimerDataSet[6].control[2].run )
   END_RUNG
   RUNG wire#w1
      { S7_Templates := "SrcType := DInt" } EQ_Contact(in1 := "Unit1.Em5.HmiInterface".mainPnP.jobs.status.activeJobNumber, in2 := "U1EM5_JOB03")
      Coil( "ProdDataInterfaceHmi".cycleTimerDataSet[6].control[3].run )
   END_RUNG
   RUNG wire#w1
      { S7_Templates := "SrcType := DInt" } EQ_Contact(in1 := "Unit1.Em5.HmiInterface".mainPnP.jobs.status.activeJobNumber, in2 := "U1EM5_JOB04")
      Coil( "ProdDataInterfaceHmi".cycleTimerDataSet[6].control[4].run )
   END_RUNG
   RUNG wire#w1
      { S7_Templates := "SrcType := DInt" } EQ_Contact(in1 := "Unit1.Em5.HmiInterface".mainPnP.jobs.status.activeJobNumber, in2 := "U1EM5_JOB05")
      Coil( "ProdDataInterfaceHmi".cycleTimerDataSet[6].control[5].run )
   END_RUNG
   RUNG wire#w1
      { S7_Templates := "SrcType := DInt" } EQ_Contact(in1 := "Unit1.Em5.HmiInterface".mainPnP.jobs.status.activeJobNumber, in2 := "U1EM5_JOB06")
      Coil( "ProdDataInterfaceHmi".cycleTimerDataSet[6].control[6].run )
   END_RUNG
   RUNG wire#w1
      { S7_Templates := "SrcType := DInt" } EQ_Contact(in1 := "Unit1.Em5.HmiInterface".mainPnP.jobs.status.activeJobNumber, in2 := "U1EM5_JOB10")
      Coil( "ProdDataInterfaceHmi".cycleTimerDataSet[6].control[8].run )
   END_RUNG
   RUNG wire#powerrail
      Contact( #TRUE )
      wire#w2
      { S7_Templates := "SrcType := DInt" } EQ_Contact(in1 := "Unit1.Em5.HmiInterface".alignTable.jobs.status.activeJobNumber, in2 := "U1EM4_JOB01")
      Coil( "ProdDataInterfaceHmi".cycleTimerDataSet[6].control[9].run )
   END_RUNG
   RUNG wire#w2
      { S7_Templates := "SrcType := DInt" } EQ_Contact(in1 := "Unit1.Em5.HmiInterface".alignTable.jobs.status.activeJobNumber, in2 := "U1EM4_JOB02")
      Coil( "ProdDataInterfaceHmi".cycleTimerDataSet[6].control[10].run )
   END_RUNG
   RUNG wire#w2
      { S7_Templates := "SrcType := DInt" } EQ_Contact(in1 := "Unit1.Em5.HmiInterface".alignTable.jobs.status.activeJobNumber, in2 := "U1EM4_JOB03")
      Coil( "ProdDataInterfaceHmi".cycleTimerDataSet[6].control[11].run )
   END_RUNG
   RUNG wire#w2
      { S7_Templates := "SrcType := DInt" } EQ_Contact(in1 := "Unit1.Em5.HmiInterface".alignTable.jobs.status.activeJobNumber, in2 := "U1EM4_JOB04")
      Coil( "ProdDataInterfaceHmi".cycleTimerDataSet[6].control[12].run )
   END_RUNG
   RUNG wire#w2
      { S7_Templates := "SrcType := DInt" } EQ_Contact(in1 := "Unit1.Em5.HmiInterface".alignTable.jobs.status.activeJobNumber, in2 := "U1EM4_JOB22")
      Coil( "ProdDataInterfaceHmi".cycleTimerDataSet[6].control[13].run )
   END_RUNG
   RUNG wire#powerrail
      Contact( #TRUE )
      wire#w3
      { S7_Templates := "SrcType := DInt" } EQ_Contact(in1 := "Unit1.Em5.HmiInterface".ngPnP.jobs.status.activeJobNumber, in2 := "U1EM4_JOB01")
      Coil( "ProdDataInterfaceHmi".cycleTimerDataSet[6].control[14].run )
   END_RUNG
   RUNG wire#w3
      { S7_Templates := "SrcType := DInt" } EQ_Contact(in1 := "Unit1.Em5.HmiInterface".ngPnP.jobs.status.activeJobNumber, in2 := "U1EM4_JOB02")
      Coil( "ProdDataInterfaceHmi".cycleTimerDataSet[6].control[15].run )
   END_RUNG
   RUNG wire#w3
      { S7_Templates := "SrcType := DInt" } EQ_Contact(in1 := "Unit1.Em5.HmiInterface".ngPnP.jobs.status.activeJobNumber, in2 := "U1EM4_JOB03")
      Coil( "ProdDataInterfaceHmi".cycleTimerDataSet[6].control[16].run )
   END_RUNG
   RUNG wire#powerrail
      Contact( #TRUE )
      { S7_Templates := "SrcType := DInt" } EQ_Contact(in1 := "Unit1.Em5.HmiInterface".gaugeRnR.jobs.status.activeJobNumber, in2 := "U1EM4_JOB01")
      Coil( "ProdDataInterfaceHmi".cycleTimerDataSet[6].control[17].run )
   END_RUNG
   // the same network as SCL:
   "ProdDataInterfaceHmi".cycleTimerDataSet[6].control[1].run := #TRUE AND ("Unit1.Em5.HmiInterface".mainPnP.jobs.status.activeJobNumber = "U1EM5_JOB01");
   "ProdDataInterfaceHmi".cycleTimerDataSet[6].control[2].run := #TRUE AND ("Unit1.Em5.HmiInterface".mainPnP.jobs.status.activeJobNumber = "U1EM5_JOB02");
   "ProdDataInterfaceHmi".cycleTimerDataSet[6].control[3].run := #TRUE AND ("Unit1.Em5.HmiInterface".mainPnP.jobs.status.activeJobNumber = "U1EM5_JOB03");
   "ProdDataInterfaceHmi".cycleTimerDataSet[6].control[4].run := #TRUE AND ("Unit1.Em5.HmiInterface".mainPnP.jobs.status.activeJobNumber = "U1EM5_JOB04");
   "ProdDataInterfaceHmi".cycleTimerDataSet[6].control[5].run := #TRUE AND ("Unit1.Em5.HmiInterface".mainPnP.jobs.status.activeJobNumber = "U1EM5_JOB05");
   "ProdDataInterfaceHmi".cycleTimerDataSet[6].control[6].run := #TRUE AND ("Unit1.Em5.HmiInterface".mainPnP.jobs.status.activeJobNumber = "U1EM5_JOB06");
   "ProdDataInterfaceHmi".cycleTimerDataSet[6].control[8].run := #TRUE AND ("Unit1.Em5.HmiInterface".mainPnP.jobs.status.activeJobNumber = "U1EM5_JOB10");
   "ProdDataInterfaceHmi".cycleTimerDataSet[6].control[9].run := #TRUE AND ("Unit1.Em5.HmiInterface".alignTable.jobs.status.activeJobNumber = "U1EM4_JOB01");
   "ProdDataInterfaceHmi".cycleTimerDataSet[6].control[10].run := #TRUE AND ("Unit1.Em5.HmiInterface".alignTable.jobs.status.activeJobNumber = "U1EM4_JOB02");
   "ProdDataInterfaceHmi".cycleTimerDataSet[6].control[11].run := #TRUE AND ("Unit1.Em5.HmiInterface".alignTable.jobs.status.activeJobNumber = "U1EM4_JOB03");
   "ProdDataInterfaceHmi".cycleTimerDataSet[6].control[12].run := #TRUE AND ("Unit1.Em5.HmiInterface".alignTable.jobs.status.activeJobNumber = "U1EM4_JOB04");
   "ProdDataInterfaceHmi".cycleTimerDataSet[6].control[13].run := #TRUE AND ("Unit1.Em5.HmiInterface".alignTable.jobs.status.activeJobNumber = "U1EM4_JOB22");
   "ProdDataInterfaceHmi".cycleTimerDataSet[6].control[14].run := #TRUE AND ("Unit1.Em5.HmiInterface".ngPnP.jobs.status.activeJobNumber = "U1EM4_JOB01");
   "ProdDataInterfaceHmi".cycleTimerDataSet[6].control[15].run := #TRUE AND ("Unit1.Em5.HmiInterface".ngPnP.jobs.status.activeJobNumber = "U1EM4_JOB02");
   "ProdDataInterfaceHmi".cycleTimerDataSet[6].control[16].run := #TRUE AND ("Unit1.Em5.HmiInterface".ngPnP.jobs.status.activeJobNumber = "U1EM4_JOB03");
   "ProdDataInterfaceHmi".cycleTimerDataSet[6].control[17].run := #TRUE AND ("Unit1.Em5.HmiInterface".gaugeRnR.jobs.status.activeJobNumber = "U1EM4_JOB01");
END_REGION

REGION Network 7: Cycle Timer Em 6
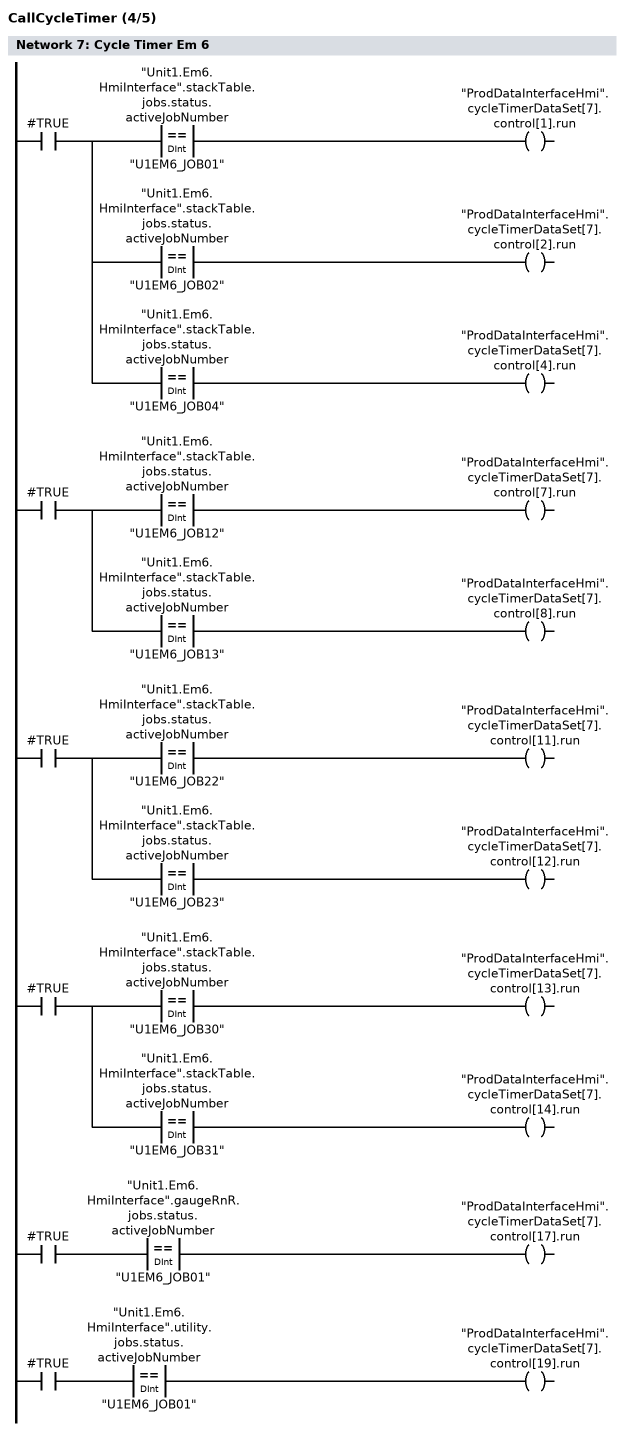
   RUNG wire#powerrail
      Contact( #TRUE )
      wire#w1
      { S7_Templates := "SrcType := DInt" } EQ_Contact(in1 := "Unit1.Em6.HmiInterface".stackTable.jobs.status.activeJobNumber, in2 := "U1EM6_JOB01")
      Coil( "ProdDataInterfaceHmi".cycleTimerDataSet[7].control[1].run )
   END_RUNG
   RUNG wire#w1
      { S7_Templates := "SrcType := DInt" } EQ_Contact(in1 := "Unit1.Em6.HmiInterface".stackTable.jobs.status.activeJobNumber, in2 := "U1EM6_JOB02")
      Coil( "ProdDataInterfaceHmi".cycleTimerDataSet[7].control[2].run )
   END_RUNG
   RUNG wire#w1
      { S7_Templates := "SrcType := DInt" } EQ_Contact(in1 := "Unit1.Em6.HmiInterface".stackTable.jobs.status.activeJobNumber, in2 := "U1EM6_JOB04")
      Coil( "ProdDataInterfaceHmi".cycleTimerDataSet[7].control[4].run )
   END_RUNG
   RUNG wire#powerrail
      Contact( #TRUE )
      wire#w2
      { S7_Templates := "SrcType := DInt" } EQ_Contact(in1 := "Unit1.Em6.HmiInterface".stackTable.jobs.status.activeJobNumber, in2 := "U1EM6_JOB12")
      Coil( "ProdDataInterfaceHmi".cycleTimerDataSet[7].control[7].run )
   END_RUNG
   RUNG wire#w2
      { S7_Templates := "SrcType := DInt" } EQ_Contact(in1 := "Unit1.Em6.HmiInterface".stackTable.jobs.status.activeJobNumber, in2 := "U1EM6_JOB13")
      Coil( "ProdDataInterfaceHmi".cycleTimerDataSet[7].control[8].run )
   END_RUNG
   RUNG wire#powerrail
      Contact( #TRUE )
      wire#w3
      { S7_Templates := "SrcType := DInt" } EQ_Contact(in1 := "Unit1.Em6.HmiInterface".stackTable.jobs.status.activeJobNumber, in2 := "U1EM6_JOB22")
      Coil( "ProdDataInterfaceHmi".cycleTimerDataSet[7].control[11].run )
   END_RUNG
   RUNG wire#w3
      { S7_Templates := "SrcType := DInt" } EQ_Contact(in1 := "Unit1.Em6.HmiInterface".stackTable.jobs.status.activeJobNumber, in2 := "U1EM6_JOB23")
      Coil( "ProdDataInterfaceHmi".cycleTimerDataSet[7].control[12].run )
   END_RUNG
   RUNG wire#powerrail
      Contact( #TRUE )
      wire#w4
      { S7_Templates := "SrcType := DInt" } EQ_Contact(in1 := "Unit1.Em6.HmiInterface".stackTable.jobs.status.activeJobNumber, in2 := "U1EM6_JOB30")
      Coil( "ProdDataInterfaceHmi".cycleTimerDataSet[7].control[13].run )
   END_RUNG
   RUNG wire#w4
      { S7_Templates := "SrcType := DInt" } EQ_Contact(in1 := "Unit1.Em6.HmiInterface".stackTable.jobs.status.activeJobNumber, in2 := "U1EM6_JOB31")
      Coil( "ProdDataInterfaceHmi".cycleTimerDataSet[7].control[14].run )
   END_RUNG
   RUNG wire#powerrail
      Contact( #TRUE )
      { S7_Templates := "SrcType := DInt" } EQ_Contact(in1 := "Unit1.Em6.HmiInterface".gaugeRnR.jobs.status.activeJobNumber, in2 := "U1EM6_JOB01")
      Coil( "ProdDataInterfaceHmi".cycleTimerDataSet[7].control[17].run )
   END_RUNG
   RUNG wire#powerrail
      Contact( #TRUE )
      { S7_Templates := "SrcType := DInt" } EQ_Contact(in1 := "Unit1.Em6.HmiInterface".utility.jobs.status.activeJobNumber, in2 := "U1EM6_JOB01")
      Coil( "ProdDataInterfaceHmi".cycleTimerDataSet[7].control[19].run )
   END_RUNG
   // the same network as SCL:
   "ProdDataInterfaceHmi".cycleTimerDataSet[7].control[1].run := #TRUE AND ("Unit1.Em6.HmiInterface".stackTable.jobs.status.activeJobNumber = "U1EM6_JOB01");
   "ProdDataInterfaceHmi".cycleTimerDataSet[7].control[2].run := #TRUE AND ("Unit1.Em6.HmiInterface".stackTable.jobs.status.activeJobNumber = "U1EM6_JOB02");
   "ProdDataInterfaceHmi".cycleTimerDataSet[7].control[4].run := #TRUE AND ("Unit1.Em6.HmiInterface".stackTable.jobs.status.activeJobNumber = "U1EM6_JOB04");
   "ProdDataInterfaceHmi".cycleTimerDataSet[7].control[7].run := #TRUE AND ("Unit1.Em6.HmiInterface".stackTable.jobs.status.activeJobNumber = "U1EM6_JOB12");
   "ProdDataInterfaceHmi".cycleTimerDataSet[7].control[8].run := #TRUE AND ("Unit1.Em6.HmiInterface".stackTable.jobs.status.activeJobNumber = "U1EM6_JOB13");
   "ProdDataInterfaceHmi".cycleTimerDataSet[7].control[11].run := #TRUE AND ("Unit1.Em6.HmiInterface".stackTable.jobs.status.activeJobNumber = "U1EM6_JOB22");
   "ProdDataInterfaceHmi".cycleTimerDataSet[7].control[12].run := #TRUE AND ("Unit1.Em6.HmiInterface".stackTable.jobs.status.activeJobNumber = "U1EM6_JOB23");
   "ProdDataInterfaceHmi".cycleTimerDataSet[7].control[13].run := #TRUE AND ("Unit1.Em6.HmiInterface".stackTable.jobs.status.activeJobNumber = "U1EM6_JOB30");
   "ProdDataInterfaceHmi".cycleTimerDataSet[7].control[14].run := #TRUE AND ("Unit1.Em6.HmiInterface".stackTable.jobs.status.activeJobNumber = "U1EM6_JOB31");
   "ProdDataInterfaceHmi".cycleTimerDataSet[7].control[17].run := #TRUE AND ("Unit1.Em6.HmiInterface".gaugeRnR.jobs.status.activeJobNumber = "U1EM6_JOB01");
   "ProdDataInterfaceHmi".cycleTimerDataSet[7].control[19].run := #TRUE AND ("Unit1.Em6.HmiInterface".utility.jobs.status.activeJobNumber = "U1EM6_JOB01");
END_REGION

REGION Network 8: Cycle Timer Em 7
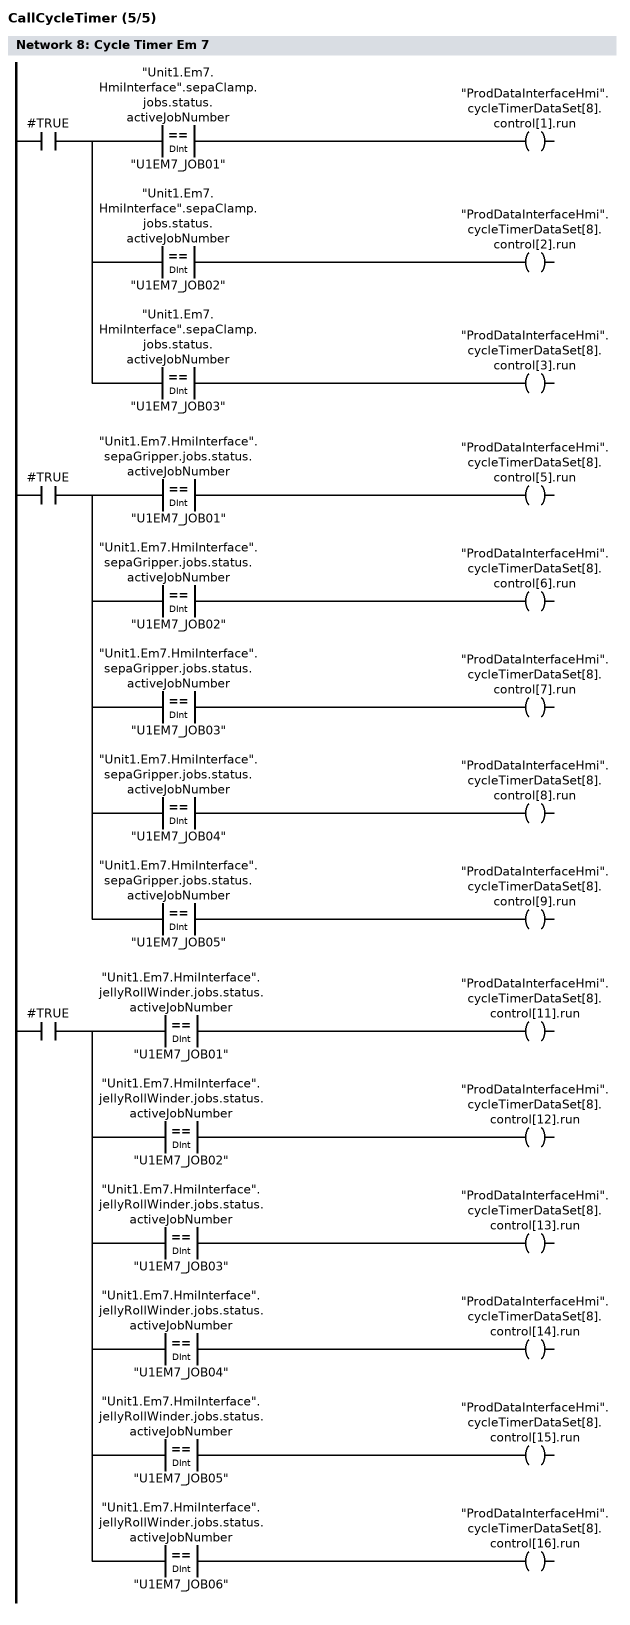
   RUNG wire#powerrail
      Contact( #TRUE )
      wire#w1
      { S7_Templates := "SrcType := DInt" } EQ_Contact(in1 := "Unit1.Em7.HmiInterface".sepaClamp.jobs.status.activeJobNumber, in2 := "U1EM7_JOB01")
      Coil( "ProdDataInterfaceHmi".cycleTimerDataSet[8].control[1].run )
   END_RUNG
   RUNG wire#w1
      { S7_Templates := "SrcType := DInt" } EQ_Contact(in1 := "Unit1.Em7.HmiInterface".sepaClamp.jobs.status.activeJobNumber, in2 := "U1EM7_JOB02")
      Coil( "ProdDataInterfaceHmi".cycleTimerDataSet[8].control[2].run )
   END_RUNG
   RUNG wire#w1
      { S7_Templates := "SrcType := DInt" } EQ_Contact(in1 := "Unit1.Em7.HmiInterface".sepaClamp.jobs.status.activeJobNumber, in2 := "U1EM7_JOB03")
      Coil( "ProdDataInterfaceHmi".cycleTimerDataSet[8].control[3].run )
   END_RUNG
   RUNG wire#powerrail
      Contact( #TRUE )
      wire#w2
      { S7_Templates := "SrcType := DInt" } EQ_Contact(in1 := "Unit1.Em7.HmiInterface".sepaGripper.jobs.status.activeJobNumber, in2 := "U1EM7_JOB01")
      Coil( "ProdDataInterfaceHmi".cycleTimerDataSet[8].control[5].run )
   END_RUNG
   RUNG wire#w2
      { S7_Templates := "SrcType := DInt" } EQ_Contact(in1 := "Unit1.Em7.HmiInterface".sepaGripper.jobs.status.activeJobNumber, in2 := "U1EM7_JOB02")
      Coil( "ProdDataInterfaceHmi".cycleTimerDataSet[8].control[6].run )
   END_RUNG
   RUNG wire#w2
      { S7_Templates := "SrcType := DInt" } EQ_Contact(in1 := "Unit1.Em7.HmiInterface".sepaGripper.jobs.status.activeJobNumber, in2 := "U1EM7_JOB03")
      Coil( "ProdDataInterfaceHmi".cycleTimerDataSet[8].control[7].run )
   END_RUNG
   RUNG wire#w2
      { S7_Templates := "SrcType := DInt" } EQ_Contact(in1 := "Unit1.Em7.HmiInterface".sepaGripper.jobs.status.activeJobNumber, in2 := "U1EM7_JOB04")
      Coil( "ProdDataInterfaceHmi".cycleTimerDataSet[8].control[8].run )
   END_RUNG
   RUNG wire#w2
      { S7_Templates := "SrcType := DInt" } EQ_Contact(in1 := "Unit1.Em7.HmiInterface".sepaGripper.jobs.status.activeJobNumber, in2 := "U1EM7_JOB05")
      Coil( "ProdDataInterfaceHmi".cycleTimerDataSet[8].control[9].run )
   END_RUNG
   RUNG wire#powerrail
      Contact( #TRUE )
      wire#w3
      { S7_Templates := "SrcType := DInt" } EQ_Contact(in1 := "Unit1.Em7.HmiInterface".jellyRollWinder.jobs.status.activeJobNumber, in2 := "U1EM7_JOB01")
      Coil( "ProdDataInterfaceHmi".cycleTimerDataSet[8].control[11].run )
   END_RUNG
   RUNG wire#w3
      { S7_Templates := "SrcType := DInt" } EQ_Contact(in1 := "Unit1.Em7.HmiInterface".jellyRollWinder.jobs.status.activeJobNumber, in2 := "U1EM7_JOB02")
      Coil( "ProdDataInterfaceHmi".cycleTimerDataSet[8].control[12].run )
   END_RUNG
   RUNG wire#w3
      { S7_Templates := "SrcType := DInt" } EQ_Contact(in1 := "Unit1.Em7.HmiInterface".jellyRollWinder.jobs.status.activeJobNumber, in2 := "U1EM7_JOB03")
      Coil( "ProdDataInterfaceHmi".cycleTimerDataSet[8].control[13].run )
   END_RUNG
   RUNG wire#w3
      { S7_Templates := "SrcType := DInt" } EQ_Contact(in1 := "Unit1.Em7.HmiInterface".jellyRollWinder.jobs.status.activeJobNumber, in2 := "U1EM7_JOB04")
      Coil( "ProdDataInterfaceHmi".cycleTimerDataSet[8].control[14].run )
   END_RUNG
   RUNG wire#w3
      { S7_Templates := "SrcType := DInt" } EQ_Contact(in1 := "Unit1.Em7.HmiInterface".jellyRollWinder.jobs.status.activeJobNumber, in2 := "U1EM7_JOB05")
      Coil( "ProdDataInterfaceHmi".cycleTimerDataSet[8].control[15].run )
   END_RUNG
   RUNG wire#w3
      { S7_Templates := "SrcType := DInt" } EQ_Contact(in1 := "Unit1.Em7.HmiInterface".jellyRollWinder.jobs.status.activeJobNumber, in2 := "U1EM7_JOB06")
      Coil( "ProdDataInterfaceHmi".cycleTimerDataSet[8].control[16].run )
   END_RUNG
   // the same network as SCL:
   "ProdDataInterfaceHmi".cycleTimerDataSet[8].control[1].run := #TRUE AND ("Unit1.Em7.HmiInterface".sepaClamp.jobs.status.activeJobNumber = "U1EM7_JOB01");
   "ProdDataInterfaceHmi".cycleTimerDataSet[8].control[2].run := #TRUE AND ("Unit1.Em7.HmiInterface".sepaClamp.jobs.status.activeJobNumber = "U1EM7_JOB02");
   "ProdDataInterfaceHmi".cycleTimerDataSet[8].control[3].run := #TRUE AND ("Unit1.Em7.HmiInterface".sepaClamp.jobs.status.activeJobNumber = "U1EM7_JOB03");
   "ProdDataInterfaceHmi".cycleTimerDataSet[8].control[5].run := #TRUE AND ("Unit1.Em7.HmiInterface".sepaGripper.jobs.status.activeJobNumber = "U1EM7_JOB01");
   "ProdDataInterfaceHmi".cycleTimerDataSet[8].control[6].run := #TRUE AND ("Unit1.Em7.HmiInterface".sepaGripper.jobs.status.activeJobNumber = "U1EM7_JOB02");
   "ProdDataInterfaceHmi".cycleTimerDataSet[8].control[7].run := #TRUE AND ("Unit1.Em7.HmiInterface".sepaGripper.jobs.status.activeJobNumber = "U1EM7_JOB03");
   "ProdDataInterfaceHmi".cycleTimerDataSet[8].control[8].run := #TRUE AND ("Unit1.Em7.HmiInterface".sepaGripper.jobs.status.activeJobNumber = "U1EM7_JOB04");
   "ProdDataInterfaceHmi".cycleTimerDataSet[8].control[9].run := #TRUE AND ("Unit1.Em7.HmiInterface".sepaGripper.jobs.status.activeJobNumber = "U1EM7_JOB05");
   "ProdDataInterfaceHmi".cycleTimerDataSet[8].control[11].run := #TRUE AND ("Unit1.Em7.HmiInterface".jellyRollWinder.jobs.status.activeJobNumber = "U1EM7_JOB01");
   "ProdDataInterfaceHmi".cycleTimerDataSet[8].control[12].run := #TRUE AND ("Unit1.Em7.HmiInterface".jellyRollWinder.jobs.status.activeJobNumber = "U1EM7_JOB02");
   "ProdDataInterfaceHmi".cycleTimerDataSet[8].control[13].run := #TRUE AND ("Unit1.Em7.HmiInterface".jellyRollWinder.jobs.status.activeJobNumber = "U1EM7_JOB03");
   "ProdDataInterfaceHmi".cycleTimerDataSet[8].control[14].run := #TRUE AND ("Unit1.Em7.HmiInterface".jellyRollWinder.jobs.status.activeJobNumber = "U1EM7_JOB04");
   "ProdDataInterfaceHmi".cycleTimerDataSet[8].control[15].run := #TRUE AND ("Unit1.Em7.HmiInterface".jellyRollWinder.jobs.status.activeJobNumber = "U1EM7_JOB05");
   "ProdDataInterfaceHmi".cycleTimerDataSet[8].control[16].run := #TRUE AND ("Unit1.Em7.HmiInterface".jellyRollWinder.jobs.status.activeJobNumber = "U1EM7_JOB06");
END_REGION
END_FUNCTION

